	WY11609_00 AT  %MX11636.0 : BOOL; (*STN 5 PROCESS TANK VACUUM RELEASE AV5-2 (-161Y10) *)
	WY11609_01 AT  %MX11636.1 : BOOL; (*STN 5 PROCESS TANK VACUUM RELEASE AV5-2 (-161Y10) *)
	WY11609_02 AT  %MX11636.2 : BOOL; (*STN 5 PROCESS TANK VACUUM RELEASE AV5-2 (-161Y10) *)
	WY11609_03 AT  %MX11636.3 : BOOL; (*STN 5 PROCESS TANK VACUUM RELEASE AV5-2 (-161Y10) *)
	WY11609_04 AT  %MX11636.4 : BOOL; (*STN 5 PROCESS TANK VACUUM RELEASE AV5-2 (-161Y10) *)
	WY11609_05 AT  %MX11636.5 : BOOL; (*STN 5 PROCESS TANK VACUUM RELEASE AV5-2 (-161Y10) *)
	WY11609_06 AT  %MX11636.6 : BOOL; (*STN 5 PROCESS TANK VACUUM RELEASE AV5-2 (-161Y10) *)
	WY11609_07 AT  %MX11636.7 : BOOL; (*STN 5 PROCESS TANK VACUUM RELEASE AV5-2 (-161Y10) *)
	WY11609_08 AT  %MX11636.8 : BOOL; (*STN 5 PROCESS TANK VACUUM RELEASE AV5-2 (-161Y10) *)
	WY11609_09 AT  %MX11636.9 : BOOL; (*STN 5 PROCESS TANK VACUUM RELEASE AV5-2 (-161Y10) *)
	WY11609_10 AT  %MX11636.10 : BOOL; (*STN 5 PROCESS TANK VACUUM RELEASE AV5-2 (-161Y10) *)
	WY11609_11 AT  %MX11636.11 : BOOL; (*STN 5 PROCESS TANK VACUUM RELEASE AV5-2 (-161Y10) *)
	WY11609_12 AT  %MX11636.12 : BOOL; (*STN 5 PROCESS TANK VACUUM RELEASE AV5-2 (-161Y10) *)
	WY11609_13 AT  %MX11636.13 : BOOL; (*STN 5 PROCESS TANK VACUUM RELEASE AV5-2 (-161Y10) *)
	WY11609_14 AT  %MX11636.14 : BOOL; (*STN 5 PROCESS TANK VACUUM RELEASE AV5-2 (-161Y10) *)
	WY11609_15 AT  %MX11636.15 : BOOL; (*STN 5 PROCESS TANK VACUUM RELEASE AV5-2 (-161Y10) *)
	WY11609_16 AT  %MX11636.16 : BOOL; (*STN 5 PROCESS TANK VACUUM RELEASE AV5-2 (-161Y10) *)
	WY11609_17 AT  %MX11636.17 : BOOL; (*STN 5 PROCESS TANK VACUUM RELEASE AV5-2 (-161Y10) *)
	WY11609_18 AT  %MX11636.18 : BOOL; (*STN 5 PROCESS TANK VACUUM RELEASE AV5-2 (-161Y10) *)
	WY11609_19 AT  %MX11636.19 : BOOL; (*STN 5 PROCESS TANK VACUUM RELEASE AV5-2 (-161Y10) *)
	WY11609_20 AT  %MX11636.20 : BOOL; (*STN 5 PROCESS TANK VACUUM RELEASE AV5-2 (-161Y10) *)
	WY11609_21 AT  %MX11636.21 : BOOL; (*STN 5 PROCESS TANK VACUUM RELEASE AV5-2 (-161Y10) *)
	WY11609_22 AT  %MX11636.22 : BOOL; (*STN 5 PROCESS TANK VACUUM RELEASE AV5-2 (-161Y10) *)
	WY11609_23 AT  %MX11636.23 : BOOL; (*STN 5 PROCESS TANK VACUUM RELEASE AV5-2 (-161Y10) *)
	WY11609_24 AT  %MX11636.24 : BOOL; (*STN 5 PROCESS TANK VACUUM RELEASE AV5-2 (-161Y10) *)
	WY11609_25 AT  %MX11636.25 : BOOL; (*STN 5 PROCESS TANK VACUUM RELEASE AV5-2 (-161Y10) *)
	WY11609_26 AT  %MX11636.26 : BOOL; (*STN 5 PROCESS TANK VACUUM RELEASE AV5-2 (-161Y10) *)
	WY11609_27 AT  %MX11636.27 : BOOL; (*STN 5 PROCESS TANK VACUUM RELEASE AV5-2 (-161Y10) *)
	WY11609_28 AT  %MX11636.28 : BOOL; (*STN 5 PROCESS TANK VACUUM RELEASE AV5-2 (-161Y10) *)
	WY11609_29 AT  %MX11636.29 : BOOL; (*STN 5 PROCESS TANK VACUUM RELEASE AV5-2 (-161Y10) *)
	WY11609_30 AT  %MX11636.30 : BOOL; (*STN 5 PROCESS TANK VACUUM RELEASE AV5-2 (-161Y10) *)
	WY11609_31 AT  %MX11636.31 : BOOL; (*STN 5 PROCESS TANK VACUUM RELEASE AV5-2 (-161Y10) *)

	WY11610_00 AT  %MX11640.0 : BOOL; (*STN 5 BLOWER PROTECTION BUTTLEFLY AV5-3 (-161Y11) *)
	WY11610_01 AT  %MX11640.1 : BOOL; (*STN 5 BLOWER PROTECTION BUTTLEFLY AV5-3 (-161Y11) *)
	WY11610_02 AT  %MX11640.2 : BOOL; (*STN 5 BLOWER PROTECTION BUTTLEFLY AV5-3 (-161Y11) *)
	WY11610_03 AT  %MX11640.3 : BOOL; (*STN 5 BLOWER PROTECTION BUTTLEFLY AV5-3 (-161Y11) *)
	WY11610_04 AT  %MX11640.4 : BOOL; (*STN 5 BLOWER PROTECTION BUTTLEFLY AV5-3 (-161Y11) *)
	WY11610_05 AT  %MX11640.5 : BOOL; (*STN 5 BLOWER PROTECTION BUTTLEFLY AV5-3 (-161Y11) *)
	WY11610_06 AT  %MX11640.6 : BOOL; (*STN 5 BLOWER PROTECTION BUTTLEFLY AV5-3 (-161Y11) *)
	WY11610_07 AT  %MX11640.7 : BOOL; (*STN 5 BLOWER PROTECTION BUTTLEFLY AV5-3 (-161Y11) *)
	WY11610_08 AT  %MX11640.8 : BOOL; (*STN 5 BLOWER PROTECTION BUTTLEFLY AV5-3 (-161Y11) *)
	WY11610_09 AT  %MX11640.9 : BOOL; (*STN 5 BLOWER PROTECTION BUTTLEFLY AV5-3 (-161Y11) *)
	WY11610_10 AT  %MX11640.10 : BOOL; (*STN 5 BLOWER PROTECTION BUTTLEFLY AV5-3 (-161Y11) *)
	WY11610_11 AT  %MX11640.11 : BOOL; (*STN 5 BLOWER PROTECTION BUTTLEFLY AV5-3 (-161Y11) *)
	WY11610_12 AT  %MX11640.12 : BOOL; (*STN 5 BLOWER PROTECTION BUTTLEFLY AV5-3 (-161Y11) *)
	WY11610_13 AT  %MX11640.13 : BOOL; (*STN 5 BLOWER PROTECTION BUTTLEFLY AV5-3 (-161Y11) *)
	WY11610_14 AT  %MX11640.14 : BOOL; (*STN 5 BLOWER PROTECTION BUTTLEFLY AV5-3 (-161Y11) *)
	WY11610_15 AT  %MX11640.15 : BOOL; (*STN 5 BLOWER PROTECTION BUTTLEFLY AV5-3 (-161Y11) *)
	WY11610_16 AT  %MX11640.16 : BOOL; (*STN 5 BLOWER PROTECTION BUTTLEFLY AV5-3 (-161Y11) *)
	WY11610_17 AT  %MX11640.17 : BOOL; (*STN 5 BLOWER PROTECTION BUTTLEFLY AV5-3 (-161Y11) *)
	WY11610_18 AT  %MX11640.18 : BOOL; (*STN 5 BLOWER PROTECTION BUTTLEFLY AV5-3 (-161Y11) *)
	WY11610_19 AT  %MX11640.19 : BOOL; (*STN 5 BLOWER PROTECTION BUTTLEFLY AV5-3 (-161Y11) *)
	WY11610_20 AT  %MX11640.20 : BOOL; (*STN 5 BLOWER PROTECTION BUTTLEFLY AV5-3 (-161Y11) *)
	WY11610_21 AT  %MX11640.21 : BOOL; (*STN 5 BLOWER PROTECTION BUTTLEFLY AV5-3 (-161Y11) *)
	WY11610_22 AT  %MX11640.22 : BOOL; (*STN 5 BLOWER PROTECTION BUTTLEFLY AV5-3 (-161Y11) *)
	WY11610_23 AT  %MX11640.23 : BOOL; (*STN 5 BLOWER PROTECTION BUTTLEFLY AV5-3 (-161Y11) *)
	WY11610_24 AT  %MX11640.24 : BOOL; (*STN 5 BLOWER PROTECTION BUTTLEFLY AV5-3 (-161Y11) *)
	WY11610_25 AT  %MX11640.25 : BOOL; (*STN 5 BLOWER PROTECTION BUTTLEFLY AV5-3 (-161Y11) *)
	WY11610_26 AT  %MX11640.26 : BOOL; (*STN 5 BLOWER PROTECTION BUTTLEFLY AV5-3 (-161Y11) *)
	WY11610_27 AT  %MX11640.27 : BOOL; (*STN 5 BLOWER PROTECTION BUTTLEFLY AV5-3 (-161Y11) *)
	WY11610_28 AT  %MX11640.28 : BOOL; (*STN 5 BLOWER PROTECTION BUTTLEFLY AV5-3 (-161Y11) *)
	WY11610_29 AT  %MX11640.29 : BOOL; (*STN 5 BLOWER PROTECTION BUTTLEFLY AV5-3 (-161Y11) *)
	WY11610_30 AT  %MX11640.30 : BOOL; (*STN 5 BLOWER PROTECTION BUTTLEFLY AV5-3 (-161Y11) *)
	WY11610_31 AT  %MX11640.31 : BOOL; (*STN 5 BLOWER PROTECTION BUTTLEFLY AV5-3 (-161Y11) *)

	WY11611_00 AT  %MX11644.0 : BOOL; (*STN 5 BLOWER PROTECTION BUTTLEFLY AV5-4 (-161Y12) *)
	WY11611_01 AT  %MX11644.1 : BOOL; (*STN 5 BLOWER PROTECTION BUTTLEFLY AV5-4 (-161Y12) *)
	WY11611_02 AT  %MX11644.2 : BOOL; (*STN 5 BLOWER PROTECTION BUTTLEFLY AV5-4 (-161Y12) *)
	WY11611_03 AT  %MX11644.3 : BOOL; (*STN 5 BLOWER PROTECTION BUTTLEFLY AV5-4 (-161Y12) *)
	WY11611_04 AT  %MX11644.4 : BOOL; (*STN 5 BLOWER PROTECTION BUTTLEFLY AV5-4 (-161Y12) *)
	WY11611_05 AT  %MX11644.5 : BOOL; (*STN 5 BLOWER PROTECTION BUTTLEFLY AV5-4 (-161Y12) *)
	WY11611_06 AT  %MX11644.6 : BOOL; (*STN 5 BLOWER PROTECTION BUTTLEFLY AV5-4 (-161Y12) *)
	WY11611_07 AT  %MX11644.7 : BOOL; (*STN 5 BLOWER PROTECTION BUTTLEFLY AV5-4 (-161Y12) *)
	WY11611_08 AT  %MX11644.8 : BOOL; (*STN 5 BLOWER PROTECTION BUTTLEFLY AV5-4 (-161Y12) *)
	WY11611_09 AT  %MX11644.9 : BOOL; (*STN 5 BLOWER PROTECTION BUTTLEFLY AV5-4 (-161Y12) *)
	WY11611_10 AT  %MX11644.10 : BOOL; (*STN 5 BLOWER PROTECTION BUTTLEFLY AV5-4 (-161Y12) *)
	WY11611_11 AT  %MX11644.11 : BOOL; (*STN 5 BLOWER PROTECTION BUTTLEFLY AV5-4 (-161Y12) *)
	WY11611_12 AT  %MX11644.12 : BOOL; (*STN 5 BLOWER PROTECTION BUTTLEFLY AV5-4 (-161Y12) *)
	WY11611_13 AT  %MX11644.13 : BOOL; (*STN 5 BLOWER PROTECTION BUTTLEFLY AV5-4 (-161Y12) *)
	WY11611_14 AT  %MX11644.14 : BOOL; (*STN 5 BLOWER PROTECTION BUTTLEFLY AV5-4 (-161Y12) *)
	WY11611_15 AT  %MX11644.15 : BOOL; (*STN 5 BLOWER PROTECTION BUTTLEFLY AV5-4 (-161Y12) *)
	WY11611_16 AT  %MX11644.16 : BOOL; (*STN 5 BLOWER PROTECTION BUTTLEFLY AV5-4 (-161Y12) *)
	WY11611_17 AT  %MX11644.17 : BOOL; (*STN 5 BLOWER PROTECTION BUTTLEFLY AV5-4 (-161Y12) *)
	WY11611_18 AT  %MX11644.18 : BOOL; (*STN 5 BLOWER PROTECTION BUTTLEFLY AV5-4 (-161Y12) *)
	WY11611_19 AT  %MX11644.19 : BOOL; (*STN 5 BLOWER PROTECTION BUTTLEFLY AV5-4 (-161Y12) *)
	WY11611_20 AT  %MX11644.20 : BOOL; (*STN 5 BLOWER PROTECTION BUTTLEFLY AV5-4 (-161Y12) *)
	WY11611_21 AT  %MX11644.21 : BOOL; (*STN 5 BLOWER PROTECTION BUTTLEFLY AV5-4 (-161Y12) *)
	WY11611_22 AT  %MX11644.22 : BOOL; (*STN 5 BLOWER PROTECTION BUTTLEFLY AV5-4 (-161Y12) *)
	WY11611_23 AT  %MX11644.23 : BOOL; (*STN 5 BLOWER PROTECTION BUTTLEFLY AV5-4 (-161Y12) *)
	WY11611_24 AT  %MX11644.24 : BOOL; (*STN 5 BLOWER PROTECTION BUTTLEFLY AV5-4 (-161Y12) *)
	WY11611_25 AT  %MX11644.25 : BOOL; (*STN 5 BLOWER PROTECTION BUTTLEFLY AV5-4 (-161Y12) *)
	WY11611_26 AT  %MX11644.26 : BOOL; (*STN 5 BLOWER PROTECTION BUTTLEFLY AV5-4 (-161Y12) *)
	WY11611_27 AT  %MX11644.27 : BOOL; (*STN 5 BLOWER PROTECTION BUTTLEFLY AV5-4 (-161Y12) *)
	WY11611_28 AT  %MX11644.28 : BOOL; (*STN 5 BLOWER PROTECTION BUTTLEFLY AV5-4 (-161Y12) *)
	WY11611_29 AT  %MX11644.29 : BOOL; (*STN 5 BLOWER PROTECTION BUTTLEFLY AV5-4 (-161Y12) *)
	WY11611_30 AT  %MX11644.30 : BOOL; (*STN 5 BLOWER PROTECTION BUTTLEFLY AV5-4 (-161Y12) *)
	WY11611_31 AT  %MX11644.31 : BOOL; (*STN 5 BLOWER PROTECTION BUTTLEFLY AV5-4 (-161Y12) *)

	WY11612_00 AT  %MX11648.0 : BOOL; (*FACILITY CHILL WATER SUPPLY AV5-5 (-161Y13) *)
	WY11612_01 AT  %MX11648.1 : BOOL; (*FACILITY CHILL WATER SUPPLY AV5-5 (-161Y13) *)
	WY11612_02 AT  %MX11648.2 : BOOL; (*FACILITY CHILL WATER SUPPLY AV5-5 (-161Y13) *)
	WY11612_03 AT  %MX11648.3 : BOOL; (*FACILITY CHILL WATER SUPPLY AV5-5 (-161Y13) *)
	WY11612_04 AT  %MX11648.4 : BOOL; (*FACILITY CHILL WATER SUPPLY AV5-5 (-161Y13) *)
	WY11612_05 AT  %MX11648.5 : BOOL; (*FACILITY CHILL WATER SUPPLY AV5-5 (-161Y13) *)
	WY11612_06 AT  %MX11648.6 : BOOL; (*FACILITY CHILL WATER SUPPLY AV5-5 (-161Y13) *)
	WY11612_07 AT  %MX11648.7 : BOOL; (*FACILITY CHILL WATER SUPPLY AV5-5 (-161Y13) *)
	WY11612_08 AT  %MX11648.8 : BOOL; (*FACILITY CHILL WATER SUPPLY AV5-5 (-161Y13) *)
	WY11612_09 AT  %MX11648.9 : BOOL; (*FACILITY CHILL WATER SUPPLY AV5-5 (-161Y13) *)
	WY11612_10 AT  %MX11648.10 : BOOL; (*FACILITY CHILL WATER SUPPLY AV5-5 (-161Y13) *)
	WY11612_11 AT  %MX11648.11 : BOOL; (*FACILITY CHILL WATER SUPPLY AV5-5 (-161Y13) *)
	WY11612_12 AT  %MX11648.12 : BOOL; (*FACILITY CHILL WATER SUPPLY AV5-5 (-161Y13) *)
	WY11612_13 AT  %MX11648.13 : BOOL; (*FACILITY CHILL WATER SUPPLY AV5-5 (-161Y13) *)
	WY11612_14 AT  %MX11648.14 : BOOL; (*FACILITY CHILL WATER SUPPLY AV5-5 (-161Y13) *)
	WY11612_15 AT  %MX11648.15 : BOOL; (*FACILITY CHILL WATER SUPPLY AV5-5 (-161Y13) *)
	WY11612_16 AT  %MX11648.16 : BOOL; (*FACILITY CHILL WATER SUPPLY AV5-5 (-161Y13) *)
	WY11612_17 AT  %MX11648.17 : BOOL; (*FACILITY CHILL WATER SUPPLY AV5-5 (-161Y13) *)
	WY11612_18 AT  %MX11648.18 : BOOL; (*FACILITY CHILL WATER SUPPLY AV5-5 (-161Y13) *)
	WY11612_19 AT  %MX11648.19 : BOOL; (*FACILITY CHILL WATER SUPPLY AV5-5 (-161Y13) *)
	WY11612_20 AT  %MX11648.20 : BOOL; (*FACILITY CHILL WATER SUPPLY AV5-5 (-161Y13) *)
	WY11612_21 AT  %MX11648.21 : BOOL; (*FACILITY CHILL WATER SUPPLY AV5-5 (-161Y13) *)
	WY11612_22 AT  %MX11648.22 : BOOL; (*FACILITY CHILL WATER SUPPLY AV5-5 (-161Y13) *)
	WY11612_23 AT  %MX11648.23 : BOOL; (*FACILITY CHILL WATER SUPPLY AV5-5 (-161Y13) *)
	WY11612_24 AT  %MX11648.24 : BOOL; (*FACILITY CHILL WATER SUPPLY AV5-5 (-161Y13) *)
	WY11612_25 AT  %MX11648.25 : BOOL; (*FACILITY CHILL WATER SUPPLY AV5-5 (-161Y13) *)
	WY11612_26 AT  %MX11648.26 : BOOL; (*FACILITY CHILL WATER SUPPLY AV5-5 (-161Y13) *)
	WY11612_27 AT  %MX11648.27 : BOOL; (*FACILITY CHILL WATER SUPPLY AV5-5 (-161Y13) *)
	WY11612_28 AT  %MX11648.28 : BOOL; (*FACILITY CHILL WATER SUPPLY AV5-5 (-161Y13) *)
	WY11612_29 AT  %MX11648.29 : BOOL; (*FACILITY CHILL WATER SUPPLY AV5-5 (-161Y13) *)
	WY11612_30 AT  %MX11648.30 : BOOL; (*FACILITY CHILL WATER SUPPLY AV5-5 (-161Y13) *)
	WY11612_31 AT  %MX11648.31 : BOOL; (*FACILITY CHILL WATER SUPPLY AV5-5 (-161Y13) *)

	WY11613_00 AT  %MX11652.0 : BOOL; (*STN 4 & UNLOADING IONIZER CDA DISCHARGE AVION-1 (-161Y14,15) *)
	WY11613_01 AT  %MX11652.1 : BOOL; (*STN 4 & UNLOADING IONIZER CDA DISCHARGE AVION-1 (-161Y14,15) *)
	WY11613_02 AT  %MX11652.2 : BOOL; (*STN 4 & UNLOADING IONIZER CDA DISCHARGE AVION-1 (-161Y14,15) *)
	WY11613_03 AT  %MX11652.3 : BOOL; (*STN 4 & UNLOADING IONIZER CDA DISCHARGE AVION-1 (-161Y14,15) *)
	WY11613_04 AT  %MX11652.4 : BOOL; (*STN 4 & UNLOADING IONIZER CDA DISCHARGE AVION-1 (-161Y14,15) *)
	WY11613_05 AT  %MX11652.5 : BOOL; (*STN 4 & UNLOADING IONIZER CDA DISCHARGE AVION-1 (-161Y14,15) *)
	WY11613_06 AT  %MX11652.6 : BOOL; (*STN 4 & UNLOADING IONIZER CDA DISCHARGE AVION-1 (-161Y14,15) *)
	WY11613_07 AT  %MX11652.7 : BOOL; (*STN 4 & UNLOADING IONIZER CDA DISCHARGE AVION-1 (-161Y14,15) *)
	WY11613_08 AT  %MX11652.8 : BOOL; (*STN 4 & UNLOADING IONIZER CDA DISCHARGE AVION-1 (-161Y14,15) *)
	WY11613_09 AT  %MX11652.9 : BOOL; (*STN 4 & UNLOADING IONIZER CDA DISCHARGE AVION-1 (-161Y14,15) *)
	WY11613_10 AT  %MX11652.10 : BOOL; (*STN 4 & UNLOADING IONIZER CDA DISCHARGE AVION-1 (-161Y14,15) *)
	WY11613_11 AT  %MX11652.11 : BOOL; (*STN 4 & UNLOADING IONIZER CDA DISCHARGE AVION-1 (-161Y14,15) *)
	WY11613_12 AT  %MX11652.12 : BOOL; (*STN 4 & UNLOADING IONIZER CDA DISCHARGE AVION-1 (-161Y14,15) *)
	WY11613_13 AT  %MX11652.13 : BOOL; (*STN 4 & UNLOADING IONIZER CDA DISCHARGE AVION-1 (-161Y14,15) *)
	WY11613_14 AT  %MX11652.14 : BOOL; (*STN 4 & UNLOADING IONIZER CDA DISCHARGE AVION-1 (-161Y14,15) *)
	WY11613_15 AT  %MX11652.15 : BOOL; (*STN 4 & UNLOADING IONIZER CDA DISCHARGE AVION-1 (-161Y14,15) *)
	WY11613_16 AT  %MX11652.16 : BOOL; (*STN 4 & UNLOADING IONIZER CDA DISCHARGE AVION-1 (-161Y14,15) *)
	WY11613_17 AT  %MX11652.17 : BOOL; (*STN 4 & UNLOADING IONIZER CDA DISCHARGE AVION-1 (-161Y14,15) *)
	WY11613_18 AT  %MX11652.18 : BOOL; (*STN 4 & UNLOADING IONIZER CDA DISCHARGE AVION-1 (-161Y14,15) *)
	WY11613_19 AT  %MX11652.19 : BOOL; (*STN 4 & UNLOADING IONIZER CDA DISCHARGE AVION-1 (-161Y14,15) *)
	WY11613_20 AT  %MX11652.20 : BOOL; (*STN 4 & UNLOADING IONIZER CDA DISCHARGE AVION-1 (-161Y14,15) *)
	WY11613_21 AT  %MX11652.21 : BOOL; (*STN 4 & UNLOADING IONIZER CDA DISCHARGE AVION-1 (-161Y14,15) *)
	WY11613_22 AT  %MX11652.22 : BOOL; (*STN 4 & UNLOADING IONIZER CDA DISCHARGE AVION-1 (-161Y14,15) *)
	WY11613_23 AT  %MX11652.23 : BOOL; (*STN 4 & UNLOADING IONIZER CDA DISCHARGE AVION-1 (-161Y14,15) *)
	WY11613_24 AT  %MX11652.24 : BOOL; (*STN 4 & UNLOADING IONIZER CDA DISCHARGE AVION-1 (-161Y14,15) *)
	WY11613_25 AT  %MX11652.25 : BOOL; (*STN 4 & UNLOADING IONIZER CDA DISCHARGE AVION-1 (-161Y14,15) *)
	WY11613_26 AT  %MX11652.26 : BOOL; (*STN 4 & UNLOADING IONIZER CDA DISCHARGE AVION-1 (-161Y14,15) *)
	WY11613_27 AT  %MX11652.27 : BOOL; (*STN 4 & UNLOADING IONIZER CDA DISCHARGE AVION-1 (-161Y14,15) *)
	WY11613_28 AT  %MX11652.28 : BOOL; (*STN 4 & UNLOADING IONIZER CDA DISCHARGE AVION-1 (-161Y14,15) *)
	WY11613_29 AT  %MX11652.29 : BOOL; (*STN 4 & UNLOADING IONIZER CDA DISCHARGE AVION-1 (-161Y14,15) *)
	WY11613_30 AT  %MX11652.30 : BOOL; (*STN 4 & UNLOADING IONIZER CDA DISCHARGE AVION-1 (-161Y14,15) *)
	WY11613_31 AT  %MX11652.31 : BOOL; (*STN 4 & UNLOADING IONIZER CDA DISCHARGE AVION-1 (-161Y14,15) *)

	WY11614_00 AT  %MX11656.0 : BOOL; (*STN 4 IONIZER STATIC ELIMINATION STOP SIGNAL (-161U1) *)
	WY11614_01 AT  %MX11656.1 : BOOL; (*STN 4 IONIZER STATIC ELIMINATION STOP SIGNAL (-161U1) *)
	WY11614_02 AT  %MX11656.2 : BOOL; (*STN 4 IONIZER STATIC ELIMINATION STOP SIGNAL (-161U1) *)
	WY11614_03 AT  %MX11656.3 : BOOL; (*STN 4 IONIZER STATIC ELIMINATION STOP SIGNAL (-161U1) *)
	WY11614_04 AT  %MX11656.4 : BOOL; (*STN 4 IONIZER STATIC ELIMINATION STOP SIGNAL (-161U1) *)
	WY11614_05 AT  %MX11656.5 : BOOL; (*STN 4 IONIZER STATIC ELIMINATION STOP SIGNAL (-161U1) *)
	WY11614_06 AT  %MX11656.6 : BOOL; (*STN 4 IONIZER STATIC ELIMINATION STOP SIGNAL (-161U1) *)
	WY11614_07 AT  %MX11656.7 : BOOL; (*STN 4 IONIZER STATIC ELIMINATION STOP SIGNAL (-161U1) *)
	WY11614_08 AT  %MX11656.8 : BOOL; (*STN 4 IONIZER STATIC ELIMINATION STOP SIGNAL (-161U1) *)
	WY11614_09 AT  %MX11656.9 : BOOL; (*STN 4 IONIZER STATIC ELIMINATION STOP SIGNAL (-161U1) *)
	WY11614_10 AT  %MX11656.10 : BOOL; (*STN 4 IONIZER STATIC ELIMINATION STOP SIGNAL (-161U1) *)
	WY11614_11 AT  %MX11656.11 : BOOL; (*STN 4 IONIZER STATIC ELIMINATION STOP SIGNAL (-161U1) *)
	WY11614_12 AT  %MX11656.12 : BOOL; (*STN 4 IONIZER STATIC ELIMINATION STOP SIGNAL (-161U1) *)
	WY11614_13 AT  %MX11656.13 : BOOL; (*STN 4 IONIZER STATIC ELIMINATION STOP SIGNAL (-161U1) *)
	WY11614_14 AT  %MX11656.14 : BOOL; (*STN 4 IONIZER STATIC ELIMINATION STOP SIGNAL (-161U1) *)
	WY11614_15 AT  %MX11656.15 : BOOL; (*STN 4 IONIZER STATIC ELIMINATION STOP SIGNAL (-161U1) *)
	WY11614_16 AT  %MX11656.16 : BOOL; (*STN 4 IONIZER STATIC ELIMINATION STOP SIGNAL (-161U1) *)
	WY11614_17 AT  %MX11656.17 : BOOL; (*STN 4 IONIZER STATIC ELIMINATION STOP SIGNAL (-161U1) *)
	WY11614_18 AT  %MX11656.18 : BOOL; (*STN 4 IONIZER STATIC ELIMINATION STOP SIGNAL (-161U1) *)
	WY11614_19 AT  %MX11656.19 : BOOL; (*STN 4 IONIZER STATIC ELIMINATION STOP SIGNAL (-161U1) *)
	WY11614_20 AT  %MX11656.20 : BOOL; (*STN 4 IONIZER STATIC ELIMINATION STOP SIGNAL (-161U1) *)
	WY11614_21 AT  %MX11656.21 : BOOL; (*STN 4 IONIZER STATIC ELIMINATION STOP SIGNAL (-161U1) *)
	WY11614_22 AT  %MX11656.22 : BOOL; (*STN 4 IONIZER STATIC ELIMINATION STOP SIGNAL (-161U1) *)
	WY11614_23 AT  %MX11656.23 : BOOL; (*STN 4 IONIZER STATIC ELIMINATION STOP SIGNAL (-161U1) *)
	WY11614_24 AT  %MX11656.24 : BOOL; (*STN 4 IONIZER STATIC ELIMINATION STOP SIGNAL (-161U1) *)
	WY11614_25 AT  %MX11656.25 : BOOL; (*STN 4 IONIZER STATIC ELIMINATION STOP SIGNAL (-161U1) *)
	WY11614_26 AT  %MX11656.26 : BOOL; (*STN 4 IONIZER STATIC ELIMINATION STOP SIGNAL (-161U1) *)
	WY11614_27 AT  %MX11656.27 : BOOL; (*STN 4 IONIZER STATIC ELIMINATION STOP SIGNAL (-161U1) *)
	WY11614_28 AT  %MX11656.28 : BOOL; (*STN 4 IONIZER STATIC ELIMINATION STOP SIGNAL (-161U1) *)
	WY11614_29 AT  %MX11656.29 : BOOL; (*STN 4 IONIZER STATIC ELIMINATION STOP SIGNAL (-161U1) *)
	WY11614_30 AT  %MX11656.30 : BOOL; (*STN 4 IONIZER STATIC ELIMINATION STOP SIGNAL (-161U1) *)
	WY11614_31 AT  %MX11656.31 : BOOL; (*STN 4 IONIZER STATIC ELIMINATION STOP SIGNAL (-161U1) *)

	WY11615_00 AT  %MX11660.0 : BOOL; (*UNLOADING IONIZER STATIC ELIMINATION STOP SIGNAL (-161U2) *)
	WY11615_01 AT  %MX11660.1 : BOOL; (*UNLOADING IONIZER STATIC ELIMINATION STOP SIGNAL (-161U2) *)
	WY11615_02 AT  %MX11660.2 : BOOL; (*UNLOADING IONIZER STATIC ELIMINATION STOP SIGNAL (-161U2) *)
	WY11615_03 AT  %MX11660.3 : BOOL; (*UNLOADING IONIZER STATIC ELIMINATION STOP SIGNAL (-161U2) *)
	WY11615_04 AT  %MX11660.4 : BOOL; (*UNLOADING IONIZER STATIC ELIMINATION STOP SIGNAL (-161U2) *)
	WY11615_05 AT  %MX11660.5 : BOOL; (*UNLOADING IONIZER STATIC ELIMINATION STOP SIGNAL (-161U2) *)
	WY11615_06 AT  %MX11660.6 : BOOL; (*UNLOADING IONIZER STATIC ELIMINATION STOP SIGNAL (-161U2) *)
	WY11615_07 AT  %MX11660.7 : BOOL; (*UNLOADING IONIZER STATIC ELIMINATION STOP SIGNAL (-161U2) *)
	WY11615_08 AT  %MX11660.8 : BOOL; (*UNLOADING IONIZER STATIC ELIMINATION STOP SIGNAL (-161U2) *)
	WY11615_09 AT  %MX11660.9 : BOOL; (*UNLOADING IONIZER STATIC ELIMINATION STOP SIGNAL (-161U2) *)
	WY11615_10 AT  %MX11660.10 : BOOL; (*UNLOADING IONIZER STATIC ELIMINATION STOP SIGNAL (-161U2) *)
	WY11615_11 AT  %MX11660.11 : BOOL; (*UNLOADING IONIZER STATIC ELIMINATION STOP SIGNAL (-161U2) *)
	WY11615_12 AT  %MX11660.12 : BOOL; (*UNLOADING IONIZER STATIC ELIMINATION STOP SIGNAL (-161U2) *)
	WY11615_13 AT  %MX11660.13 : BOOL; (*UNLOADING IONIZER STATIC ELIMINATION STOP SIGNAL (-161U2) *)
	WY11615_14 AT  %MX11660.14 : BOOL; (*UNLOADING IONIZER STATIC ELIMINATION STOP SIGNAL (-161U2) *)
	WY11615_15 AT  %MX11660.15 : BOOL; (*UNLOADING IONIZER STATIC ELIMINATION STOP SIGNAL (-161U2) *)
	WY11615_16 AT  %MX11660.16 : BOOL; (*UNLOADING IONIZER STATIC ELIMINATION STOP SIGNAL (-161U2) *)
	WY11615_17 AT  %MX11660.17 : BOOL; (*UNLOADING IONIZER STATIC ELIMINATION STOP SIGNAL (-161U2) *)
	WY11615_18 AT  %MX11660.18 : BOOL; (*UNLOADING IONIZER STATIC ELIMINATION STOP SIGNAL (-161U2) *)
	WY11615_19 AT  %MX11660.19 : BOOL; (*UNLOADING IONIZER STATIC ELIMINATION STOP SIGNAL (-161U2) *)
	WY11615_20 AT  %MX11660.20 : BOOL; (*UNLOADING IONIZER STATIC ELIMINATION STOP SIGNAL (-161U2) *)
	WY11615_21 AT  %MX11660.21 : BOOL; (*UNLOADING IONIZER STATIC ELIMINATION STOP SIGNAL (-161U2) *)
	WY11615_22 AT  %MX11660.22 : BOOL; (*UNLOADING IONIZER STATIC ELIMINATION STOP SIGNAL (-161U2) *)
	WY11615_23 AT  %MX11660.23 : BOOL; (*UNLOADING IONIZER STATIC ELIMINATION STOP SIGNAL (-161U2) *)
	WY11615_24 AT  %MX11660.24 : BOOL; (*UNLOADING IONIZER STATIC ELIMINATION STOP SIGNAL (-161U2) *)
	WY11615_25 AT  %MX11660.25 : BOOL; (*UNLOADING IONIZER STATIC ELIMINATION STOP SIGNAL (-161U2) *)
	WY11615_26 AT  %MX11660.26 : BOOL; (*UNLOADING IONIZER STATIC ELIMINATION STOP SIGNAL (-161U2) *)
	WY11615_27 AT  %MX11660.27 : BOOL; (*UNLOADING IONIZER STATIC ELIMINATION STOP SIGNAL (-161U2) *)
	WY11615_28 AT  %MX11660.28 : BOOL; (*UNLOADING IONIZER STATIC ELIMINATION STOP SIGNAL (-161U2) *)
	WY11615_29 AT  %MX11660.29 : BOOL; (*UNLOADING IONIZER STATIC ELIMINATION STOP SIGNAL (-161U2) *)
	WY11615_30 AT  %MX11660.30 : BOOL; (*UNLOADING IONIZER STATIC ELIMINATION STOP SIGNAL (-161U2) *)
	WY11615_31 AT  %MX11660.31 : BOOL; (*UNLOADING IONIZER STATIC ELIMINATION STOP SIGNAL (-161U2) *)

	WY11700_00 AT  %MX11700.0 : BOOL; (*STN 4 CDA CYLINDER - IN (-162Y1) *)
	WY11700_01 AT  %MX11700.1 : BOOL; (*STN 4 CDA CYLINDER - IN (-162Y1) *)
	WY11700_02 AT  %MX11700.2 : BOOL; (*STN 4 CDA CYLINDER - IN (-162Y1) *)
	WY11700_03 AT  %MX11700.3 : BOOL; (*STN 4 CDA CYLINDER - IN (-162Y1) *)
	WY11700_04 AT  %MX11700.4 : BOOL; (*STN 4 CDA CYLINDER - IN (-162Y1) *)
	WY11700_05 AT  %MX11700.5 : BOOL; (*STN 4 CDA CYLINDER - IN (-162Y1) *)
	WY11700_06 AT  %MX11700.6 : BOOL; (*STN 4 CDA CYLINDER - IN (-162Y1) *)
	WY11700_07 AT  %MX11700.7 : BOOL; (*STN 4 CDA CYLINDER - IN (-162Y1) *)
	WY11700_08 AT  %MX11700.8 : BOOL; (*STN 4 CDA CYLINDER - IN (-162Y1) *)
	WY11700_09 AT  %MX11700.9 : BOOL; (*STN 4 CDA CYLINDER - IN (-162Y1) *)
	WY11700_10 AT  %MX11700.10 : BOOL; (*STN 4 CDA CYLINDER - IN (-162Y1) *)
	WY11700_11 AT  %MX11700.11 : BOOL; (*STN 4 CDA CYLINDER - IN (-162Y1) *)
	WY11700_12 AT  %MX11700.12 : BOOL; (*STN 4 CDA CYLINDER - IN (-162Y1) *)
	WY11700_13 AT  %MX11700.13 : BOOL; (*STN 4 CDA CYLINDER - IN (-162Y1) *)
	WY11700_14 AT  %MX11700.14 : BOOL; (*STN 4 CDA CYLINDER - IN (-162Y1) *)
	WY11700_15 AT  %MX11700.15 : BOOL; (*STN 4 CDA CYLINDER - IN (-162Y1) *)
	WY11700_16 AT  %MX11700.16 : BOOL; (*STN 4 CDA CYLINDER - IN (-162Y1) *)
	WY11700_17 AT  %MX11700.17 : BOOL; (*STN 4 CDA CYLINDER - IN (-162Y1) *)
	WY11700_18 AT  %MX11700.18 : BOOL; (*STN 4 CDA CYLINDER - IN (-162Y1) *)
	WY11700_19 AT  %MX11700.19 : BOOL; (*STN 4 CDA CYLINDER - IN (-162Y1) *)
	WY11700_20 AT  %MX11700.20 : BOOL; (*STN 4 CDA CYLINDER - IN (-162Y1) *)
	WY11700_21 AT  %MX11700.21 : BOOL; (*STN 4 CDA CYLINDER - IN (-162Y1) *)
	WY11700_22 AT  %MX11700.22 : BOOL; (*STN 4 CDA CYLINDER - IN (-162Y1) *)
	WY11700_23 AT  %MX11700.23 : BOOL; (*STN 4 CDA CYLINDER - IN (-162Y1) *)
	WY11700_24 AT  %MX11700.24 : BOOL; (*STN 4 CDA CYLINDER - IN (-162Y1) *)
	WY11700_25 AT  %MX11700.25 : BOOL; (*STN 4 CDA CYLINDER - IN (-162Y1) *)
	WY11700_26 AT  %MX11700.26 : BOOL; (*STN 4 CDA CYLINDER - IN (-162Y1) *)
	WY11700_27 AT  %MX11700.27 : BOOL; (*STN 4 CDA CYLINDER - IN (-162Y1) *)
	WY11700_28 AT  %MX11700.28 : BOOL; (*STN 4 CDA CYLINDER - IN (-162Y1) *)
	WY11700_29 AT  %MX11700.29 : BOOL; (*STN 4 CDA CYLINDER - IN (-162Y1) *)
	WY11700_30 AT  %MX11700.30 : BOOL; (*STN 4 CDA CYLINDER - IN (-162Y1) *)
	WY11700_31 AT  %MX11700.31 : BOOL; (*STN 4 CDA CYLINDER - IN (-162Y1) *)

	WY11701_00 AT  %MX11704.0 : BOOL; (*STN 4 CDA CYLINDER - OUT (-162Y2) *)
	WY11701_01 AT  %MX11704.1 : BOOL; (*STN 4 CDA CYLINDER - OUT (-162Y2) *)
	WY11701_02 AT  %MX11704.2 : BOOL; (*STN 4 CDA CYLINDER - OUT (-162Y2) *)
	WY11701_03 AT  %MX11704.3 : BOOL; (*STN 4 CDA CYLINDER - OUT (-162Y2) *)
	WY11701_04 AT  %MX11704.4 : BOOL; (*STN 4 CDA CYLINDER - OUT (-162Y2) *)
	WY11701_05 AT  %MX11704.5 : BOOL; (*STN 4 CDA CYLINDER - OUT (-162Y2) *)
	WY11701_06 AT  %MX11704.6 : BOOL; (*STN 4 CDA CYLINDER - OUT (-162Y2) *)
	WY11701_07 AT  %MX11704.7 : BOOL; (*STN 4 CDA CYLINDER - OUT (-162Y2) *)
	WY11701_08 AT  %MX11704.8 : BOOL; (*STN 4 CDA CYLINDER - OUT (-162Y2) *)
	WY11701_09 AT  %MX11704.9 : BOOL; (*STN 4 CDA CYLINDER - OUT (-162Y2) *)
	WY11701_10 AT  %MX11704.10 : BOOL; (*STN 4 CDA CYLINDER - OUT (-162Y2) *)
	WY11701_11 AT  %MX11704.11 : BOOL; (*STN 4 CDA CYLINDER - OUT (-162Y2) *)
	WY11701_12 AT  %MX11704.12 : BOOL; (*STN 4 CDA CYLINDER - OUT (-162Y2) *)
	WY11701_13 AT  %MX11704.13 : BOOL; (*STN 4 CDA CYLINDER - OUT (-162Y2) *)
	WY11701_14 AT  %MX11704.14 : BOOL; (*STN 4 CDA CYLINDER - OUT (-162Y2) *)
	WY11701_15 AT  %MX11704.15 : BOOL; (*STN 4 CDA CYLINDER - OUT (-162Y2) *)
	WY11701_16 AT  %MX11704.16 : BOOL; (*STN 4 CDA CYLINDER - OUT (-162Y2) *)
	WY11701_17 AT  %MX11704.17 : BOOL; (*STN 4 CDA CYLINDER - OUT (-162Y2) *)
	WY11701_18 AT  %MX11704.18 : BOOL; (*STN 4 CDA CYLINDER - OUT (-162Y2) *)
	WY11701_19 AT  %MX11704.19 : BOOL; (*STN 4 CDA CYLINDER - OUT (-162Y2) *)
	WY11701_20 AT  %MX11704.20 : BOOL; (*STN 4 CDA CYLINDER - OUT (-162Y2) *)
	WY11701_21 AT  %MX11704.21 : BOOL; (*STN 4 CDA CYLINDER - OUT (-162Y2) *)
	WY11701_22 AT  %MX11704.22 : BOOL; (*STN 4 CDA CYLINDER - OUT (-162Y2) *)
	WY11701_23 AT  %MX11704.23 : BOOL; (*STN 4 CDA CYLINDER - OUT (-162Y2) *)
	WY11701_24 AT  %MX11704.24 : BOOL; (*STN 4 CDA CYLINDER - OUT (-162Y2) *)
	WY11701_25 AT  %MX11704.25 : BOOL; (*STN 4 CDA CYLINDER - OUT (-162Y2) *)
	WY11701_26 AT  %MX11704.26 : BOOL; (*STN 4 CDA CYLINDER - OUT (-162Y2) *)
	WY11701_27 AT  %MX11704.27 : BOOL; (*STN 4 CDA CYLINDER - OUT (-162Y2) *)
	WY11701_28 AT  %MX11704.28 : BOOL; (*STN 4 CDA CYLINDER - OUT (-162Y2) *)
	WY11701_29 AT  %MX11704.29 : BOOL; (*STN 4 CDA CYLINDER - OUT (-162Y2) *)
	WY11701_30 AT  %MX11704.30 : BOOL; (*STN 4 CDA CYLINDER - OUT (-162Y2) *)
	WY11701_31 AT  %MX11704.31 : BOOL; (*STN 4 CDA CYLINDER - OUT (-162Y2) *)

	WY11702_00 AT  %MX11708.0 : BOOL; (*RAMP PUMP AV (-162Y3) *)
	WY11702_01 AT  %MX11708.1 : BOOL; (*RAMP PUMP AV (-162Y3) *)
	WY11702_02 AT  %MX11708.2 : BOOL; (*RAMP PUMP AV (-162Y3) *)
	WY11702_03 AT  %MX11708.3 : BOOL; (*RAMP PUMP AV (-162Y3) *)
	WY11702_04 AT  %MX11708.4 : BOOL; (*RAMP PUMP AV (-162Y3) *)
	WY11702_05 AT  %MX11708.5 : BOOL; (*RAMP PUMP AV (-162Y3) *)
	WY11702_06 AT  %MX11708.6 : BOOL; (*RAMP PUMP AV (-162Y3) *)
	WY11702_07 AT  %MX11708.7 : BOOL; (*RAMP PUMP AV (-162Y3) *)
	WY11702_08 AT  %MX11708.8 : BOOL; (*RAMP PUMP AV (-162Y3) *)
	WY11702_09 AT  %MX11708.9 : BOOL; (*RAMP PUMP AV (-162Y3) *)
	WY11702_10 AT  %MX11708.10 : BOOL; (*RAMP PUMP AV (-162Y3) *)
	WY11702_11 AT  %MX11708.11 : BOOL; (*RAMP PUMP AV (-162Y3) *)
	WY11702_12 AT  %MX11708.12 : BOOL; (*RAMP PUMP AV (-162Y3) *)
	WY11702_13 AT  %MX11708.13 : BOOL; (*RAMP PUMP AV (-162Y3) *)
	WY11702_14 AT  %MX11708.14 : BOOL; (*RAMP PUMP AV (-162Y3) *)
	WY11702_15 AT  %MX11708.15 : BOOL; (*RAMP PUMP AV (-162Y3) *)
	WY11702_16 AT  %MX11708.16 : BOOL; (*RAMP PUMP AV (-162Y3) *)
	WY11702_17 AT  %MX11708.17 : BOOL; (*RAMP PUMP AV (-162Y3) *)
	WY11702_18 AT  %MX11708.18 : BOOL; (*RAMP PUMP AV (-162Y3) *)
	WY11702_19 AT  %MX11708.19 : BOOL; (*RAMP PUMP AV (-162Y3) *)
	WY11702_20 AT  %MX11708.20 : BOOL; (*RAMP PUMP AV (-162Y3) *)
	WY11702_21 AT  %MX11708.21 : BOOL; (*RAMP PUMP AV (-162Y3) *)
	WY11702_22 AT  %MX11708.22 : BOOL; (*RAMP PUMP AV (-162Y3) *)
	WY11702_23 AT  %MX11708.23 : BOOL; (*RAMP PUMP AV (-162Y3) *)
	WY11702_24 AT  %MX11708.24 : BOOL; (*RAMP PUMP AV (-162Y3) *)
	WY11702_25 AT  %MX11708.25 : BOOL; (*RAMP PUMP AV (-162Y3) *)
	WY11702_26 AT  %MX11708.26 : BOOL; (*RAMP PUMP AV (-162Y3) *)
	WY11702_27 AT  %MX11708.27 : BOOL; (*RAMP PUMP AV (-162Y3) *)
	WY11702_28 AT  %MX11708.28 : BOOL; (*RAMP PUMP AV (-162Y3) *)
	WY11702_29 AT  %MX11708.29 : BOOL; (*RAMP PUMP AV (-162Y3) *)
	WY11702_30 AT  %MX11708.30 : BOOL; (*RAMP PUMP AV (-162Y3) *)
	WY11702_31 AT  %MX11708.31 : BOOL; (*RAMP PUMP AV (-162Y3) *)

	WY11703_00 AT  %MX11712.0 : BOOL; (*RESERVED *)
	WY11703_01 AT  %MX11712.1 : BOOL; (*RESERVED *)
	WY11703_02 AT  %MX11712.2 : BOOL; (*RESERVED *)
	WY11703_03 AT  %MX11712.3 : BOOL; (*RESERVED *)
	WY11703_04 AT  %MX11712.4 : BOOL; (*RESERVED *)
	WY11703_05 AT  %MX11712.5 : BOOL; (*RESERVED *)
	WY11703_06 AT  %MX11712.6 : BOOL; (*RESERVED *)
	WY11703_07 AT  %MX11712.7 : BOOL; (*RESERVED *)
	WY11703_08 AT  %MX11712.8 : BOOL; (*RESERVED *)
	WY11703_09 AT  %MX11712.9 : BOOL; (*RESERVED *)
	WY11703_10 AT  %MX11712.10 : BOOL; (*RESERVED *)
	WY11703_11 AT  %MX11712.11 : BOOL; (*RESERVED *)
	WY11703_12 AT  %MX11712.12 : BOOL; (*RESERVED *)
	WY11703_13 AT  %MX11712.13 : BOOL; (*RESERVED *)
	WY11703_14 AT  %MX11712.14 : BOOL; (*RESERVED *)
	WY11703_15 AT  %MX11712.15 : BOOL; (*RESERVED *)
	WY11703_16 AT  %MX11712.16 : BOOL; (*RESERVED *)
	WY11703_17 AT  %MX11712.17 : BOOL; (*RESERVED *)
	WY11703_18 AT  %MX11712.18 : BOOL; (*RESERVED *)
	WY11703_19 AT  %MX11712.19 : BOOL; (*RESERVED *)
	WY11703_20 AT  %MX11712.20 : BOOL; (*RESERVED *)
	WY11703_21 AT  %MX11712.21 : BOOL; (*RESERVED *)
	WY11703_22 AT  %MX11712.22 : BOOL; (*RESERVED *)
	WY11703_23 AT  %MX11712.23 : BOOL; (*RESERVED *)
	WY11703_24 AT  %MX11712.24 : BOOL; (*RESERVED *)
	WY11703_25 AT  %MX11712.25 : BOOL; (*RESERVED *)
	WY11703_26 AT  %MX11712.26 : BOOL; (*RESERVED *)
	WY11703_27 AT  %MX11712.27 : BOOL; (*RESERVED *)
	WY11703_28 AT  %MX11712.28 : BOOL; (*RESERVED *)
	WY11703_29 AT  %MX11712.29 : BOOL; (*RESERVED *)
	WY11703_30 AT  %MX11712.30 : BOOL; (*RESERVED *)
	WY11703_31 AT  %MX11712.31 : BOOL; (*RESERVED *)

	WY11704_00 AT  %MX11716.0 : BOOL; (*RESERVED *)
	WY11704_01 AT  %MX11716.1 : BOOL; (*RESERVED *)
	WY11704_02 AT  %MX11716.2 : BOOL; (*RESERVED *)
	WY11704_03 AT  %MX11716.3 : BOOL; (*RESERVED *)
	WY11704_04 AT  %MX11716.4 : BOOL; (*RESERVED *)
	WY11704_05 AT  %MX11716.5 : BOOL; (*RESERVED *)
	WY11704_06 AT  %MX11716.6 : BOOL; (*RESERVED *)
	WY11704_07 AT  %MX11716.7 : BOOL; (*RESERVED *)
	WY11704_08 AT  %MX11716.8 : BOOL; (*RESERVED *)
	WY11704_09 AT  %MX11716.9 : BOOL; (*RESERVED *)
	WY11704_10 AT  %MX11716.10 : BOOL; (*RESERVED *)
	WY11704_11 AT  %MX11716.11 : BOOL; (*RESERVED *)
	WY11704_12 AT  %MX11716.12 : BOOL; (*RESERVED *)
	WY11704_13 AT  %MX11716.13 : BOOL; (*RESERVED *)
	WY11704_14 AT  %MX11716.14 : BOOL; (*RESERVED *)
	WY11704_15 AT  %MX11716.15 : BOOL; (*RESERVED *)
	WY11704_16 AT  %MX11716.16 : BOOL; (*RESERVED *)
	WY11704_17 AT  %MX11716.17 : BOOL; (*RESERVED *)
	WY11704_18 AT  %MX11716.18 : BOOL; (*RESERVED *)
	WY11704_19 AT  %MX11716.19 : BOOL; (*RESERVED *)
	WY11704_20 AT  %MX11716.20 : BOOL; (*RESERVED *)
	WY11704_21 AT  %MX11716.21 : BOOL; (*RESERVED *)
	WY11704_22 AT  %MX11716.22 : BOOL; (*RESERVED *)
	WY11704_23 AT  %MX11716.23 : BOOL; (*RESERVED *)
	WY11704_24 AT  %MX11716.24 : BOOL; (*RESERVED *)
	WY11704_25 AT  %MX11716.25 : BOOL; (*RESERVED *)
	WY11704_26 AT  %MX11716.26 : BOOL; (*RESERVED *)
	WY11704_27 AT  %MX11716.27 : BOOL; (*RESERVED *)
	WY11704_28 AT  %MX11716.28 : BOOL; (*RESERVED *)
	WY11704_29 AT  %MX11716.29 : BOOL; (*RESERVED *)
	WY11704_30 AT  %MX11716.30 : BOOL; (*RESERVED *)
	WY11704_31 AT  %MX11716.31 : BOOL; (*RESERVED *)

	WY11705_00 AT  %MX11720.0 : BOOL; (*RESERVED *)
	WY11705_01 AT  %MX11720.1 : BOOL; (*RESERVED *)
	WY11705_02 AT  %MX11720.2 : BOOL; (*RESERVED *)
	WY11705_03 AT  %MX11720.3 : BOOL; (*RESERVED *)
	WY11705_04 AT  %MX11720.4 : BOOL; (*RESERVED *)
	WY11705_05 AT  %MX11720.5 : BOOL; (*RESERVED *)
	WY11705_06 AT  %MX11720.6 : BOOL; (*RESERVED *)
	WY11705_07 AT  %MX11720.7 : BOOL; (*RESERVED *)
	WY11705_08 AT  %MX11720.8 : BOOL; (*RESERVED *)
	WY11705_09 AT  %MX11720.9 : BOOL; (*RESERVED *)
	WY11705_10 AT  %MX11720.10 : BOOL; (*RESERVED *)
	WY11705_11 AT  %MX11720.11 : BOOL; (*RESERVED *)
	WY11705_12 AT  %MX11720.12 : BOOL; (*RESERVED *)
	WY11705_13 AT  %MX11720.13 : BOOL; (*RESERVED *)
	WY11705_14 AT  %MX11720.14 : BOOL; (*RESERVED *)
	WY11705_15 AT  %MX11720.15 : BOOL; (*RESERVED *)
	WY11705_16 AT  %MX11720.16 : BOOL; (*RESERVED *)
	WY11705_17 AT  %MX11720.17 : BOOL; (*RESERVED *)
	WY11705_18 AT  %MX11720.18 : BOOL; (*RESERVED *)
	WY11705_19 AT  %MX11720.19 : BOOL; (*RESERVED *)
	WY11705_20 AT  %MX11720.20 : BOOL; (*RESERVED *)
	WY11705_21 AT  %MX11720.21 : BOOL; (*RESERVED *)
	WY11705_22 AT  %MX11720.22 : BOOL; (*RESERVED *)
	WY11705_23 AT  %MX11720.23 : BOOL; (*RESERVED *)
	WY11705_24 AT  %MX11720.24 : BOOL; (*RESERVED *)
	WY11705_25 AT  %MX11720.25 : BOOL; (*RESERVED *)
	WY11705_26 AT  %MX11720.26 : BOOL; (*RESERVED *)
	WY11705_27 AT  %MX11720.27 : BOOL; (*RESERVED *)
	WY11705_28 AT  %MX11720.28 : BOOL; (*RESERVED *)
	WY11705_29 AT  %MX11720.29 : BOOL; (*RESERVED *)
	WY11705_30 AT  %MX11720.30 : BOOL; (*RESERVED *)
	WY11705_31 AT  %MX11720.31 : BOOL; (*RESERVED *)

	WY11706_00 AT  %MX11724.0 : BOOL; (*RESERVED *)
	WY11706_01 AT  %MX11724.1 : BOOL; (*RESERVED *)
	WY11706_02 AT  %MX11724.2 : BOOL; (*RESERVED *)
	WY11706_03 AT  %MX11724.3 : BOOL; (*RESERVED *)
	WY11706_04 AT  %MX11724.4 : BOOL; (*RESERVED *)
	WY11706_05 AT  %MX11724.5 : BOOL; (*RESERVED *)
	WY11706_06 AT  %MX11724.6 : BOOL; (*RESERVED *)
	WY11706_07 AT  %MX11724.7 : BOOL; (*RESERVED *)
	WY11706_08 AT  %MX11724.8 : BOOL; (*RESERVED *)
	WY11706_09 AT  %MX11724.9 : BOOL; (*RESERVED *)
	WY11706_10 AT  %MX11724.10 : BOOL; (*RESERVED *)
	WY11706_11 AT  %MX11724.11 : BOOL; (*RESERVED *)
	WY11706_12 AT  %MX11724.12 : BOOL; (*RESERVED *)
	WY11706_13 AT  %MX11724.13 : BOOL; (*RESERVED *)
	WY11706_14 AT  %MX11724.14 : BOOL; (*RESERVED *)
	WY11706_15 AT  %MX11724.15 : BOOL; (*RESERVED *)
	WY11706_16 AT  %MX11724.16 : BOOL; (*RESERVED *)
	WY11706_17 AT  %MX11724.17 : BOOL; (*RESERVED *)
	WY11706_18 AT  %MX11724.18 : BOOL; (*RESERVED *)
	WY11706_19 AT  %MX11724.19 : BOOL; (*RESERVED *)
	WY11706_20 AT  %MX11724.20 : BOOL; (*RESERVED *)
	WY11706_21 AT  %MX11724.21 : BOOL; (*RESERVED *)
	WY11706_22 AT  %MX11724.22 : BOOL; (*RESERVED *)
	WY11706_23 AT  %MX11724.23 : BOOL; (*RESERVED *)
	WY11706_24 AT  %MX11724.24 : BOOL; (*RESERVED *)
	WY11706_25 AT  %MX11724.25 : BOOL; (*RESERVED *)
	WY11706_26 AT  %MX11724.26 : BOOL; (*RESERVED *)
	WY11706_27 AT  %MX11724.27 : BOOL; (*RESERVED *)
	WY11706_28 AT  %MX11724.28 : BOOL; (*RESERVED *)
	WY11706_29 AT  %MX11724.29 : BOOL; (*RESERVED *)
	WY11706_30 AT  %MX11724.30 : BOOL; (*RESERVED *)
	WY11706_31 AT  %MX11724.31 : BOOL; (*RESERVED *)

	WY11707_00 AT  %MX11728.0 : BOOL; (*RESERVED *)
	WY11707_01 AT  %MX11728.1 : BOOL; (*RESERVED *)
	WY11707_02 AT  %MX11728.2 : BOOL; (*RESERVED *)
	WY11707_03 AT  %MX11728.3 : BOOL; (*RESERVED *)
	WY11707_04 AT  %MX11728.4 : BOOL; (*RESERVED *)
	WY11707_05 AT  %MX11728.5 : BOOL; (*RESERVED *)
	WY11707_06 AT  %MX11728.6 : BOOL; (*RESERVED *)
	WY11707_07 AT  %MX11728.7 : BOOL; (*RESERVED *)
	WY11707_08 AT  %MX11728.8 : BOOL; (*RESERVED *)
	WY11707_09 AT  %MX11728.9 : BOOL; (*RESERVED *)
	WY11707_10 AT  %MX11728.10 : BOOL; (*RESERVED *)
	WY11707_11 AT  %MX11728.11 : BOOL; (*RESERVED *)
	WY11707_12 AT  %MX11728.12 : BOOL; (*RESERVED *)
	WY11707_13 AT  %MX11728.13 : BOOL; (*RESERVED *)
	WY11707_14 AT  %MX11728.14 : BOOL; (*RESERVED *)
	WY11707_15 AT  %MX11728.15 : BOOL; (*RESERVED *)
	WY11707_16 AT  %MX11728.16 : BOOL; (*RESERVED *)
	WY11707_17 AT  %MX11728.17 : BOOL; (*RESERVED *)
	WY11707_18 AT  %MX11728.18 : BOOL; (*RESERVED *)
	WY11707_19 AT  %MX11728.19 : BOOL; (*RESERVED *)
	WY11707_20 AT  %MX11728.20 : BOOL; (*RESERVED *)
	WY11707_21 AT  %MX11728.21 : BOOL; (*RESERVED *)
	WY11707_22 AT  %MX11728.22 : BOOL; (*RESERVED *)
	WY11707_23 AT  %MX11728.23 : BOOL; (*RESERVED *)
	WY11707_24 AT  %MX11728.24 : BOOL; (*RESERVED *)
	WY11707_25 AT  %MX11728.25 : BOOL; (*RESERVED *)
	WY11707_26 AT  %MX11728.26 : BOOL; (*RESERVED *)
	WY11707_27 AT  %MX11728.27 : BOOL; (*RESERVED *)
	WY11707_28 AT  %MX11728.28 : BOOL; (*RESERVED *)
	WY11707_29 AT  %MX11728.29 : BOOL; (*RESERVED *)
	WY11707_30 AT  %MX11728.30 : BOOL; (*RESERVED *)
	WY11707_31 AT  %MX11728.31 : BOOL; (*RESERVED *)

	WY11708_00 AT  %MX11732.0 : BOOL; (*RESERVED *)
	WY11708_01 AT  %MX11732.1 : BOOL; (*RESERVED *)
	WY11708_02 AT  %MX11732.2 : BOOL; (*RESERVED *)
	WY11708_03 AT  %MX11732.3 : BOOL; (*RESERVED *)
	WY11708_04 AT  %MX11732.4 : BOOL; (*RESERVED *)
	WY11708_05 AT  %MX11732.5 : BOOL; (*RESERVED *)
	WY11708_06 AT  %MX11732.6 : BOOL; (*RESERVED *)
	WY11708_07 AT  %MX11732.7 : BOOL; (*RESERVED *)
	WY11708_08 AT  %MX11732.8 : BOOL; (*RESERVED *)
	WY11708_09 AT  %MX11732.9 : BOOL; (*RESERVED *)
	WY11708_10 AT  %MX11732.10 : BOOL; (*RESERVED *)
	WY11708_11 AT  %MX11732.11 : BOOL; (*RESERVED *)
	WY11708_12 AT  %MX11732.12 : BOOL; (*RESERVED *)
	WY11708_13 AT  %MX11732.13 : BOOL; (*RESERVED *)
	WY11708_14 AT  %MX11732.14 : BOOL; (*RESERVED *)
	WY11708_15 AT  %MX11732.15 : BOOL; (*RESERVED *)
	WY11708_16 AT  %MX11732.16 : BOOL; (*RESERVED *)
	WY11708_17 AT  %MX11732.17 : BOOL; (*RESERVED *)
	WY11708_18 AT  %MX11732.18 : BOOL; (*RESERVED *)
	WY11708_19 AT  %MX11732.19 : BOOL; (*RESERVED *)
	WY11708_20 AT  %MX11732.20 : BOOL; (*RESERVED *)
	WY11708_21 AT  %MX11732.21 : BOOL; (*RESERVED *)
	WY11708_22 AT  %MX11732.22 : BOOL; (*RESERVED *)
	WY11708_23 AT  %MX11732.23 : BOOL; (*RESERVED *)
	WY11708_24 AT  %MX11732.24 : BOOL; (*RESERVED *)
	WY11708_25 AT  %MX11732.25 : BOOL; (*RESERVED *)
	WY11708_26 AT  %MX11732.26 : BOOL; (*RESERVED *)
	WY11708_27 AT  %MX11732.27 : BOOL; (*RESERVED *)
	WY11708_28 AT  %MX11732.28 : BOOL; (*RESERVED *)
	WY11708_29 AT  %MX11732.29 : BOOL; (*RESERVED *)
	WY11708_30 AT  %MX11732.30 : BOOL; (*RESERVED *)
	WY11708_31 AT  %MX11732.31 : BOOL; (*RESERVED *)

	WY11709_00 AT  %MX11736.0 : BOOL; (*RESERVED *)
	WY11709_01 AT  %MX11736.1 : BOOL; (*RESERVED *)
	WY11709_02 AT  %MX11736.2 : BOOL; (*RESERVED *)
	WY11709_03 AT  %MX11736.3 : BOOL; (*RESERVED *)
	WY11709_04 AT  %MX11736.4 : BOOL; (*RESERVED *)
	WY11709_05 AT  %MX11736.5 : BOOL; (*RESERVED *)
	WY11709_06 AT  %MX11736.6 : BOOL; (*RESERVED *)
	WY11709_07 AT  %MX11736.7 : BOOL; (*RESERVED *)
	WY11709_08 AT  %MX11736.8 : BOOL; (*RESERVED *)
	WY11709_09 AT  %MX11736.9 : BOOL; (*RESERVED *)
	WY11709_10 AT  %MX11736.10 : BOOL; (*RESERVED *)
	WY11709_11 AT  %MX11736.11 : BOOL; (*RESERVED *)
	WY11709_12 AT  %MX11736.12 : BOOL; (*RESERVED *)
	WY11709_13 AT  %MX11736.13 : BOOL; (*RESERVED *)
	WY11709_14 AT  %MX11736.14 : BOOL; (*RESERVED *)
	WY11709_15 AT  %MX11736.15 : BOOL; (*RESERVED *)
	WY11709_16 AT  %MX11736.16 : BOOL; (*RESERVED *)
	WY11709_17 AT  %MX11736.17 : BOOL; (*RESERVED *)
	WY11709_18 AT  %MX11736.18 : BOOL; (*RESERVED *)
	WY11709_19 AT  %MX11736.19 : BOOL; (*RESERVED *)
	WY11709_20 AT  %MX11736.20 : BOOL; (*RESERVED *)
	WY11709_21 AT  %MX11736.21 : BOOL; (*RESERVED *)
	WY11709_22 AT  %MX11736.22 : BOOL; (*RESERVED *)
	WY11709_23 AT  %MX11736.23 : BOOL; (*RESERVED *)
	WY11709_24 AT  %MX11736.24 : BOOL; (*RESERVED *)
	WY11709_25 AT  %MX11736.25 : BOOL; (*RESERVED *)
	WY11709_26 AT  %MX11736.26 : BOOL; (*RESERVED *)
	WY11709_27 AT  %MX11736.27 : BOOL; (*RESERVED *)
	WY11709_28 AT  %MX11736.28 : BOOL; (*RESERVED *)
	WY11709_29 AT  %MX11736.29 : BOOL; (*RESERVED *)
	WY11709_30 AT  %MX11736.30 : BOOL; (*RESERVED *)
	WY11709_31 AT  %MX11736.31 : BOOL; (*RESERVED *)

	WY11710_00 AT  %MX11740.0 : BOOL; (*RESERVED *)
	WY11710_01 AT  %MX11740.1 : BOOL; (*RESERVED *)
	WY11710_02 AT  %MX11740.2 : BOOL; (*RESERVED *)
	WY11710_03 AT  %MX11740.3 : BOOL; (*RESERVED *)
	WY11710_04 AT  %MX11740.4 : BOOL; (*RESERVED *)
	WY11710_05 AT  %MX11740.5 : BOOL; (*RESERVED *)
	WY11710_06 AT  %MX11740.6 : BOOL; (*RESERVED *)
	WY11710_07 AT  %MX11740.7 : BOOL; (*RESERVED *)
	WY11710_08 AT  %MX11740.8 : BOOL; (*RESERVED *)
	WY11710_09 AT  %MX11740.9 : BOOL; (*RESERVED *)
	WY11710_10 AT  %MX11740.10 : BOOL; (*RESERVED *)
	WY11710_11 AT  %MX11740.11 : BOOL; (*RESERVED *)
	WY11710_12 AT  %MX11740.12 : BOOL; (*RESERVED *)
	WY11710_13 AT  %MX11740.13 : BOOL; (*RESERVED *)
	WY11710_14 AT  %MX11740.14 : BOOL; (*RESERVED *)
	WY11710_15 AT  %MX11740.15 : BOOL; (*RESERVED *)
	WY11710_16 AT  %MX11740.16 : BOOL; (*RESERVED *)
	WY11710_17 AT  %MX11740.17 : BOOL; (*RESERVED *)
	WY11710_18 AT  %MX11740.18 : BOOL; (*RESERVED *)
	WY11710_19 AT  %MX11740.19 : BOOL; (*RESERVED *)
	WY11710_20 AT  %MX11740.20 : BOOL; (*RESERVED *)
	WY11710_21 AT  %MX11740.21 : BOOL; (*RESERVED *)
	WY11710_22 AT  %MX11740.22 : BOOL; (*RESERVED *)
	WY11710_23 AT  %MX11740.23 : BOOL; (*RESERVED *)
	WY11710_24 AT  %MX11740.24 : BOOL; (*RESERVED *)
	WY11710_25 AT  %MX11740.25 : BOOL; (*RESERVED *)
	WY11710_26 AT  %MX11740.26 : BOOL; (*RESERVED *)
	WY11710_27 AT  %MX11740.27 : BOOL; (*RESERVED *)
	WY11710_28 AT  %MX11740.28 : BOOL; (*RESERVED *)
	WY11710_29 AT  %MX11740.29 : BOOL; (*RESERVED *)
	WY11710_30 AT  %MX11740.30 : BOOL; (*RESERVED *)
	WY11710_31 AT  %MX11740.31 : BOOL; (*RESERVED *)

	WY11711_00 AT  %MX11744.0 : BOOL; (*RESERVED *)
	WY11711_01 AT  %MX11744.1 : BOOL; (*RESERVED *)
	WY11711_02 AT  %MX11744.2 : BOOL; (*RESERVED *)
	WY11711_03 AT  %MX11744.3 : BOOL; (*RESERVED *)
	WY11711_04 AT  %MX11744.4 : BOOL; (*RESERVED *)
	WY11711_05 AT  %MX11744.5 : BOOL; (*RESERVED *)
	WY11711_06 AT  %MX11744.6 : BOOL; (*RESERVED *)
	WY11711_07 AT  %MX11744.7 : BOOL; (*RESERVED *)
	WY11711_08 AT  %MX11744.8 : BOOL; (*RESERVED *)
	WY11711_09 AT  %MX11744.9 : BOOL; (*RESERVED *)
	WY11711_10 AT  %MX11744.10 : BOOL; (*RESERVED *)
	WY11711_11 AT  %MX11744.11 : BOOL; (*RESERVED *)
	WY11711_12 AT  %MX11744.12 : BOOL; (*RESERVED *)
	WY11711_13 AT  %MX11744.13 : BOOL; (*RESERVED *)
	WY11711_14 AT  %MX11744.14 : BOOL; (*RESERVED *)
	WY11711_15 AT  %MX11744.15 : BOOL; (*RESERVED *)
	WY11711_16 AT  %MX11744.16 : BOOL; (*RESERVED *)
	WY11711_17 AT  %MX11744.17 : BOOL; (*RESERVED *)
	WY11711_18 AT  %MX11744.18 : BOOL; (*RESERVED *)
	WY11711_19 AT  %MX11744.19 : BOOL; (*RESERVED *)
	WY11711_20 AT  %MX11744.20 : BOOL; (*RESERVED *)
	WY11711_21 AT  %MX11744.21 : BOOL; (*RESERVED *)
	WY11711_22 AT  %MX11744.22 : BOOL; (*RESERVED *)
	WY11711_23 AT  %MX11744.23 : BOOL; (*RESERVED *)
	WY11711_24 AT  %MX11744.24 : BOOL; (*RESERVED *)
	WY11711_25 AT  %MX11744.25 : BOOL; (*RESERVED *)
	WY11711_26 AT  %MX11744.26 : BOOL; (*RESERVED *)
	WY11711_27 AT  %MX11744.27 : BOOL; (*RESERVED *)
	WY11711_28 AT  %MX11744.28 : BOOL; (*RESERVED *)
	WY11711_29 AT  %MX11744.29 : BOOL; (*RESERVED *)
	WY11711_30 AT  %MX11744.30 : BOOL; (*RESERVED *)
	WY11711_31 AT  %MX11744.31 : BOOL; (*RESERVED *)

	WY11712_00 AT  %MX11748.0 : BOOL; (*RESERVED *)
	WY11712_01 AT  %MX11748.1 : BOOL; (*RESERVED *)
	WY11712_02 AT  %MX11748.2 : BOOL; (*RESERVED *)
	WY11712_03 AT  %MX11748.3 : BOOL; (*RESERVED *)
	WY11712_04 AT  %MX11748.4 : BOOL; (*RESERVED *)
	WY11712_05 AT  %MX11748.5 : BOOL; (*RESERVED *)
	WY11712_06 AT  %MX11748.6 : BOOL; (*RESERVED *)
	WY11712_07 AT  %MX11748.7 : BOOL; (*RESERVED *)
	WY11712_08 AT  %MX11748.8 : BOOL; (*RESERVED *)
	WY11712_09 AT  %MX11748.9 : BOOL; (*RESERVED *)
	WY11712_10 AT  %MX11748.10 : BOOL; (*RESERVED *)
	WY11712_11 AT  %MX11748.11 : BOOL; (*RESERVED *)
	WY11712_12 AT  %MX11748.12 : BOOL; (*RESERVED *)
	WY11712_13 AT  %MX11748.13 : BOOL; (*RESERVED *)
	WY11712_14 AT  %MX11748.14 : BOOL; (*RESERVED *)
	WY11712_15 AT  %MX11748.15 : BOOL; (*RESERVED *)
	WY11712_16 AT  %MX11748.16 : BOOL; (*RESERVED *)
	WY11712_17 AT  %MX11748.17 : BOOL; (*RESERVED *)
	WY11712_18 AT  %MX11748.18 : BOOL; (*RESERVED *)
	WY11712_19 AT  %MX11748.19 : BOOL; (*RESERVED *)
	WY11712_20 AT  %MX11748.20 : BOOL; (*RESERVED *)
	WY11712_21 AT  %MX11748.21 : BOOL; (*RESERVED *)
	WY11712_22 AT  %MX11748.22 : BOOL; (*RESERVED *)
	WY11712_23 AT  %MX11748.23 : BOOL; (*RESERVED *)
	WY11712_24 AT  %MX11748.24 : BOOL; (*RESERVED *)
	WY11712_25 AT  %MX11748.25 : BOOL; (*RESERVED *)
	WY11712_26 AT  %MX11748.26 : BOOL; (*RESERVED *)
	WY11712_27 AT  %MX11748.27 : BOOL; (*RESERVED *)
	WY11712_28 AT  %MX11748.28 : BOOL; (*RESERVED *)
	WY11712_29 AT  %MX11748.29 : BOOL; (*RESERVED *)
	WY11712_30 AT  %MX11748.30 : BOOL; (*RESERVED *)
	WY11712_31 AT  %MX11748.31 : BOOL; (*RESERVED *)

	WY11713_00 AT  %MX11752.0 : BOOL; (*RESERVED *)
	WY11713_01 AT  %MX11752.1 : BOOL; (*RESERVED *)
	WY11713_02 AT  %MX11752.2 : BOOL; (*RESERVED *)
	WY11713_03 AT  %MX11752.3 : BOOL; (*RESERVED *)
	WY11713_04 AT  %MX11752.4 : BOOL; (*RESERVED *)
	WY11713_05 AT  %MX11752.5 : BOOL; (*RESERVED *)
	WY11713_06 AT  %MX11752.6 : BOOL; (*RESERVED *)
	WY11713_07 AT  %MX11752.7 : BOOL; (*RESERVED *)
	WY11713_08 AT  %MX11752.8 : BOOL; (*RESERVED *)
	WY11713_09 AT  %MX11752.9 : BOOL; (*RESERVED *)
	WY11713_10 AT  %MX11752.10 : BOOL; (*RESERVED *)
	WY11713_11 AT  %MX11752.11 : BOOL; (*RESERVED *)
	WY11713_12 AT  %MX11752.12 : BOOL; (*RESERVED *)
	WY11713_13 AT  %MX11752.13 : BOOL; (*RESERVED *)
	WY11713_14 AT  %MX11752.14 : BOOL; (*RESERVED *)
	WY11713_15 AT  %MX11752.15 : BOOL; (*RESERVED *)
	WY11713_16 AT  %MX11752.16 : BOOL; (*RESERVED *)
	WY11713_17 AT  %MX11752.17 : BOOL; (*RESERVED *)
	WY11713_18 AT  %MX11752.18 : BOOL; (*RESERVED *)
	WY11713_19 AT  %MX11752.19 : BOOL; (*RESERVED *)
	WY11713_20 AT  %MX11752.20 : BOOL; (*RESERVED *)
	WY11713_21 AT  %MX11752.21 : BOOL; (*RESERVED *)
	WY11713_22 AT  %MX11752.22 : BOOL; (*RESERVED *)
	WY11713_23 AT  %MX11752.23 : BOOL; (*RESERVED *)
	WY11713_24 AT  %MX11752.24 : BOOL; (*RESERVED *)
	WY11713_25 AT  %MX11752.25 : BOOL; (*RESERVED *)
	WY11713_26 AT  %MX11752.26 : BOOL; (*RESERVED *)
	WY11713_27 AT  %MX11752.27 : BOOL; (*RESERVED *)
	WY11713_28 AT  %MX11752.28 : BOOL; (*RESERVED *)
	WY11713_29 AT  %MX11752.29 : BOOL; (*RESERVED *)
	WY11713_30 AT  %MX11752.30 : BOOL; (*RESERVED *)
	WY11713_31 AT  %MX11752.31 : BOOL; (*RESERVED *)

	WY11714_00 AT  %MX11756.0 : BOOL; (*RESERVED *)
	WY11714_01 AT  %MX11756.1 : BOOL; (*RESERVED *)
	WY11714_02 AT  %MX11756.2 : BOOL; (*RESERVED *)
	WY11714_03 AT  %MX11756.3 : BOOL; (*RESERVED *)
	WY11714_04 AT  %MX11756.4 : BOOL; (*RESERVED *)
	WY11714_05 AT  %MX11756.5 : BOOL; (*RESERVED *)
	WY11714_06 AT  %MX11756.6 : BOOL; (*RESERVED *)
	WY11714_07 AT  %MX11756.7 : BOOL; (*RESERVED *)
	WY11714_08 AT  %MX11756.8 : BOOL; (*RESERVED *)
	WY11714_09 AT  %MX11756.9 : BOOL; (*RESERVED *)
	WY11714_10 AT  %MX11756.10 : BOOL; (*RESERVED *)
	WY11714_11 AT  %MX11756.11 : BOOL; (*RESERVED *)
	WY11714_12 AT  %MX11756.12 : BOOL; (*RESERVED *)
	WY11714_13 AT  %MX11756.13 : BOOL; (*RESERVED *)
	WY11714_14 AT  %MX11756.14 : BOOL; (*RESERVED *)
	WY11714_15 AT  %MX11756.15 : BOOL; (*RESERVED *)
	WY11714_16 AT  %MX11756.16 : BOOL; (*RESERVED *)
	WY11714_17 AT  %MX11756.17 : BOOL; (*RESERVED *)
	WY11714_18 AT  %MX11756.18 : BOOL; (*RESERVED *)
	WY11714_19 AT  %MX11756.19 : BOOL; (*RESERVED *)
	WY11714_20 AT  %MX11756.20 : BOOL; (*RESERVED *)
	WY11714_21 AT  %MX11756.21 : BOOL; (*RESERVED *)
	WY11714_22 AT  %MX11756.22 : BOOL; (*RESERVED *)
	WY11714_23 AT  %MX11756.23 : BOOL; (*RESERVED *)
	WY11714_24 AT  %MX11756.24 : BOOL; (*RESERVED *)
	WY11714_25 AT  %MX11756.25 : BOOL; (*RESERVED *)
	WY11714_26 AT  %MX11756.26 : BOOL; (*RESERVED *)
	WY11714_27 AT  %MX11756.27 : BOOL; (*RESERVED *)
	WY11714_28 AT  %MX11756.28 : BOOL; (*RESERVED *)
	WY11714_29 AT  %MX11756.29 : BOOL; (*RESERVED *)
	WY11714_30 AT  %MX11756.30 : BOOL; (*RESERVED *)
	WY11714_31 AT  %MX11756.31 : BOOL; (*RESERVED *)

	WY11715_00 AT  %MX11760.0 : BOOL; (*RESERVED *)
	WY11715_01 AT  %MX11760.1 : BOOL; (*RESERVED *)
	WY11715_02 AT  %MX11760.2 : BOOL; (*RESERVED *)
	WY11715_03 AT  %MX11760.3 : BOOL; (*RESERVED *)
	WY11715_04 AT  %MX11760.4 : BOOL; (*RESERVED *)
	WY11715_05 AT  %MX11760.5 : BOOL; (*RESERVED *)
	WY11715_06 AT  %MX11760.6 : BOOL; (*RESERVED *)
	WY11715_07 AT  %MX11760.7 : BOOL; (*RESERVED *)
	WY11715_08 AT  %MX11760.8 : BOOL; (*RESERVED *)
	WY11715_09 AT  %MX11760.9 : BOOL; (*RESERVED *)
	WY11715_10 AT  %MX11760.10 : BOOL; (*RESERVED *)
	WY11715_11 AT  %MX11760.11 : BOOL; (*RESERVED *)
	WY11715_12 AT  %MX11760.12 : BOOL; (*RESERVED *)
	WY11715_13 AT  %MX11760.13 : BOOL; (*RESERVED *)
	WY11715_14 AT  %MX11760.14 : BOOL; (*RESERVED *)
	WY11715_15 AT  %MX11760.15 : BOOL; (*RESERVED *)
	WY11715_16 AT  %MX11760.16 : BOOL; (*RESERVED *)
	WY11715_17 AT  %MX11760.17 : BOOL; (*RESERVED *)
	WY11715_18 AT  %MX11760.18 : BOOL; (*RESERVED *)
	WY11715_19 AT  %MX11760.19 : BOOL; (*RESERVED *)
	WY11715_20 AT  %MX11760.20 : BOOL; (*RESERVED *)
	WY11715_21 AT  %MX11760.21 : BOOL; (*RESERVED *)
	WY11715_22 AT  %MX11760.22 : BOOL; (*RESERVED *)
	WY11715_23 AT  %MX11760.23 : BOOL; (*RESERVED *)
	WY11715_24 AT  %MX11760.24 : BOOL; (*RESERVED *)
	WY11715_25 AT  %MX11760.25 : BOOL; (*RESERVED *)
	WY11715_26 AT  %MX11760.26 : BOOL; (*RESERVED *)
	WY11715_27 AT  %MX11760.27 : BOOL; (*RESERVED *)
	WY11715_28 AT  %MX11760.28 : BOOL; (*RESERVED *)
	WY11715_29 AT  %MX11760.29 : BOOL; (*RESERVED *)
	WY11715_30 AT  %MX11760.30 : BOOL; (*RESERVED *)
	WY11715_31 AT  %MX11760.31 : BOOL; (*RESERVED *)

END_VAR

// ---- GVLs/Digital_Ctrl/Global_Variables_DigitalMapping.TcGVL
{attribute 'Tc2GvlVarNames'}
VAR_GLOBAL

(* xxxxxxxxxxxxxxxxxxxxxxxxxxxxxxxx DIGITAL INPUT xxxxxxxxxxxxxxxxxxxxxxxxxxxxxxxx*)
(*========================================================================*)
(*
	X100_00  AT %I* : BOOL; (*GENERAL ALARM PB - RESET (-100S1)*)
	X100_01  AT %I* : BOOL; (*GENERAL BUZZER PB - RESET (-100S2)*)
	X100_02  AT %I* : BOOL; (*GENERAL MAIN PANEL PB - E-STOP (-100S3)*)
	X100_03  AT %I* : BOOL; (*OPERATOR PULL STRING - E-STOP (-100S4)*)
	X100_04  AT %I* : BOOL; (*MAINTENANCE E/STOP PULL STRING (-100S5)*)
	X100_05  AT %I* : BOOL; (*GENERAL PHASE SEQEUNCE RELAY - TRIP (-8K1)*)
	X100_06  AT %I* : BOOL; (*STN 1 PROCESS TANK PUMP TOR - TRIP (-50F2)*)
	X100_07  AT %I* : BOOL; (*STN 2 PROCESS TANK PUMP TOR - TRIP (-51F2)*)
	X100_08  AT %I* : BOOL; (*STN 3 PROCESS TANK PUMP TOR - TRIP (-52F2)*)
	X100_09  AT %I* : BOOL; (*STN 2&3 AGITATION MOTOR TOR - TRIP (-25F2)*)
	X100_10  AT %I* : BOOL; (*STN 5 BLOWER TOR - TRIP (-65F2)*)
	X100_11  AT %I* : BOOL; (*STN 5 VACUUM PUMP TOR - TRIP (-56F2)*)
	X100_12  AT %I* : BOOL; (*RESERVED*)
	X100_13  AT %I* : BOOL; (*RESERVED*)
	X100_14  AT %I* : BOOL; (*RESERVED*)
	X100_15  AT %I* : BOOL; (*RESERVED*)

	X101_00  AT %I* : BOOL; (*STN 1 SLIDING DOOR RS - OPEN (-101S5)*)
	X101_01  AT %I* : BOOL; (*STN 1 SLIDING DOOR RS - CLOSE (-101S6)*)
	X101_02  AT %I* : BOOL; (*ARM 1 HORZ SENSOR - LD SIDE OT  (-101B1)*)
	X101_03  AT %I* : BOOL; (*ARM 1 HORZ SENSOR - HOME (-101B2)*)
	X101_04  AT %I* : BOOL; (*STN 1 SUB PROCESS TANK HEATER THERMOSTAT A - ALARM (-101S8)*)
	X101_05  AT %I* : BOOL; (*STN 1 SUB PROCESS TANK HEATER THERMOSTAT B - ALARM (-101S9)*)
	X101_06  AT %I* : BOOL; (*STN 1 PROCESS TANK SENSOR - MIN LEVEL (-101S1)*)
	X101_07  AT %I* : BOOL; (*STN 1 SUB PROCESS TANK SENSOR - REG LEVEL (-101S2)*)
	X101_08  AT %I* : BOOL; (*STN 1 SUB PROCESS TANK SENSOR - MIN LEVEL (-101S3)*)
	X101_09  AT %I* : BOOL; (*DETERGENT STORAGE TANK SENSOR - MIN LEVEL (-101S4)*)
	X101_10  AT %I* : BOOL; (*STRUCTURE 1 DRIP PAN SENSOR - LEAK (-101B3)*)
	X101_11  AT %I* : BOOL; (*STN 1 SUB PROCESS TANK SENSOR - TOP UP LEVEL (-101S7)*)
	X101_12  AT %I* : BOOL; (*RESERVED*)
	X101_13  AT %I* : BOOL; (*RESERVED*)
	X101_14  AT %I* : BOOL; (*RESERVED*)
	X101_15  AT %I* : BOOL; (*RESERVED*)

	X102_00  AT %I* : BOOL; (*MODULE 1 DOOR MAGNETIC SWITCH FRONT MAINTENANCE TOP - ALARM (-102S1,2,3)*)
	X102_01  AT %I* : BOOL; (*RESERVED*)
	X102_02  AT %I* : BOOL; (*RESERVED*)
	X102_03  AT %I* : BOOL; (*MODULE 1 SLIDING DOOR SENSOR A (-102B7)*)
	X102_04  AT %I* : BOOL; (*MODULE 1 SLIDING DOOR SENSOR B (-102B8)*)
	X102_05  AT %I* : BOOL; (*RESERVED*)
	X102_06  AT %I* : BOOL; (*RESERVED*)
	X102_07  AT %I* : BOOL; (*RESERVED*)
	X102_08  AT %I* : BOOL; (*RESERVED*)
	X102_09  AT %I* : BOOL; (*RESERVED*)
	X102_10  AT %I* : BOOL; (*RESERVED*)
	X102_11  AT %I* : BOOL; (*RESERVED*)
	X102_12  AT %I* : BOOL; (*RESERVED*)
	X102_13  AT %I* : BOOL; (*RESERVED*)
	X102_14  AT %I* : BOOL; (*RESERVED*)
	X102_15  AT %I* : BOOL; (*RESERVED*)

	X110_00  AT %I* : BOOL; (*STN 2 PROCESS TANK SENSOR - MIN LEVEL (-110S1)*)
	X110_01  AT %I* : BOOL; (*STN 2 SUB PROCESS TANK SENSOR - REG LEVEL (-110S2)*)
	X110_02  AT %I* : BOOL; (*STN 2 SUB PROCESS TANK SENSOR - MIN LEVEL (-110S3)*)
	X110_03  AT %I* : BOOL; (*STN 3 PROCESS TANK SENSOR - MIN LEVEL (-110S4)*)
	X110_04  AT %I* : BOOL; (*STN 3 SUB PROCESS TANK SENSOR - REG LEVEL (-110S5)*)
	X110_05  AT %I* : BOOL; (*STN 3 SUB PROCESS TANK SENSOR - MIN LEVEL (-110S6)*)
	X110_06  AT %I* : BOOL; (*ARM 1 VERT SENSOR - TOP SIDE OT (-110B1)*)
	X110_07  AT %I* : BOOL; (*ARM 1 VERT SENSOR - TOP SIDE HOME (-110B2)*)
	X110_08  AT %I* : BOOL; (*ARM 1 VERT SENSOR - BOTTOM SIDE OT (-110B3)*)
	X110_09  AT %I* : BOOL; (*ARM 1 VERT SENSOR - CRASH (-110B4)*)
	X110_10  AT %I* : BOOL; (*ARM 1 SENSOR A - MISSHOOK (-110B5)*)
	X110_11  AT %I* : BOOL; (*ARM 1 SENSOR B - MISSHOOK (-110B6)*)
	X110_12  AT %I* : BOOL; (*RESERVED*)
	X110_13  AT %I* : BOOL; (*RESERVED*)
	X110_14  AT %I* : BOOL; (*RESERVED*)
	X110_15  AT %I* : BOOL; (*RESERVED*)

	X111_00  AT %I* : BOOL; (*STRUCTURE 2 DRIP PAN SENSOR - LEAK (-111B1)*)
	X111_01  AT %I* : BOOL; (*STN 2 SUB PROCESS TANK HEATER THERMOSTAT A - ALARM (-111S1)*)
	X111_02  AT %I* : BOOL; (*STN 2 SUB PROCESS TANK HEATER THERMOSTAT B - ALARM (-111S2)*)
	X111_03  AT %I* : BOOL; (*STN 3 SUB PROCESS TANK HEATER THERMOSTAT A - ALARM (-111S3)*)
	X111_04  AT %I* : BOOL; (*STN 3 SUB PROCESS TANK HEATER THERMOSTAT B - ALARM (-111S4)*)
	X111_05  AT %I* : BOOL; (*MODULE 2 DOOR MAGNETIC SWITCH FRONT MAINTENANCE TOP - ALARM (-111S11,12)*)
	X111_06  AT %I* : BOOL; (*RESERVED*)
	X111_07  AT %I* : BOOL; (*RESERVED*)
	X111_08  AT %I* : BOOL; (*MODULE 2 SLIDING DOOR SENSOR A (-111B2)*)
	X111_09  AT %I* : BOOL; (*MODULE 2 SLIDING DOOR SENSOR B (-111B3)*)
	X111_10  AT %I* : BOOL; (*MODULE 2 SLIDING DOOR SENSOR C (-111B4)*)
	X111_11  AT %I* : BOOL; (*RESERVED*)
	X111_12  AT %I* : BOOL; (*RESERVED*)
	X111_13  AT %I* : BOOL; (*RESERVED*)
	X111_14  AT %I* : BOOL; (*RESERVED*)
	X111_15  AT %I* : BOOL; (*RESERVED*)

	X115_00  AT %I* : BOOL; (*ARM 1 HORZ SENSOR - ULD SIDE OT (-115B1)*)
	X115_01  AT %I* : BOOL; (*ULD CONVEYOR SENSOR - FEED (-115B2)*)
	X115_02  AT %I* : BOOL; (*ULD CONVEYOR SENSOR - PICK (-115B3)*)
	X115_03  AT %I* : BOOL; (*ULD CONVEYOR PB - RAPID (-115S11)*)
	X115_04  AT %I* : BOOL; (*ULD CONVEYOR PB - E-STOP (-115S12)*)
	X115_05  AT %I* : BOOL; (*STN 4 SLIDING DOOR RS - OPEN (-115S1)*)
	X115_06  AT %I* : BOOL; (*STN 4 SLIDING DOOR RS - CLOSE (-115S2)*)
	X115_07  AT %I* : BOOL; (*STN 5 SLIDING DOOR RS - OPEN (-115S3)*)
	X115_08  AT %I* : BOOL; (*STN 5 SLIDING DOOR RS - CLOSE (-115S4)*)
	X115_09  AT %I* : BOOL; (*STN 5 SLIDING DOOR RS_A - CLAMP (-115S5)*)
	X115_10  AT %I* : BOOL; (*STN 5 SLIDING DOOR RS_A - UNCLAMP (-115S6)*)
	X115_11  AT %I* : BOOL; (*STN 5 SLIDING DOOR RS_B - CLAMP (-115S7)*)
	X115_12  AT %I* : BOOL; (*STN 5 SLIDING DOOR RS_B - UNCLAMP (-115S8)*)
	X115_13  AT %I* : BOOL; (*STN 5 PROCESS TANK HEATER THERMOSTAT - ALARM (-115S9)*)
	X115_14  AT %I* : BOOL; (*GENERAL INCOMING FLOW SENSOR - MIN FLOW (-115B4)*)
	X115_15  AT %I* : BOOL; (*RESERVED*)

	X116_00  AT %I* : BOOL; (*MAIN INC HEATER THERMOSTAT A - ALARM (-116S1)*)
	X116_01  AT %I* : BOOL; (*MAIN INC HEATER THERMOSTAT B - ALARM (-116S2)*)
	X116_02  AT %I* : BOOL; (*STN 4 IONIZER ION LEVEL ALARM (-116U1)*)
	X116_03  AT %I* : BOOL; (*STN 4 IONIZER CONDITION ALARM (-116U1)*)
	X116_04  AT %I* : BOOL; (*STN 4 IONIZER ALARM OUTPUT (-116U1)*)
	X116_05  AT %I* : BOOL; (*UNLOADING IONIZER ION LEVEL ALARM (-116U2)*)
	X116_06  AT %I* : BOOL; (*UNLOADING IONIZER CONDITION ALARM (-116U2)*)
	X116_07  AT %I* : BOOL; (*UNLOADING IONIZER ALARM OUTPUT (-116U2)*)
	X116_08  AT %I* : BOOL; (*MODULE 3 DOOR MAGNETIC SWITCH FRONT MAINTENANCE TOP - ALARM (-116S3,4,5,6,7,8,9)*)
	X116_09  AT %I* : BOOL; (*RESERVED*)
	X116_10  AT %I* : BOOL; (*RESERVED*)
	X116_11  AT %I* : BOOL; (*MODULE 3 SLIDING DOOR SENSOR A (-116B1)*)
	X116_12  AT %I* : BOOL; (*MODULE 3 SLIDING DOOR SENSOR B (-116B2)*)
	X116_13  AT %I* : BOOL; (*MODULE 3 SLIDING DOOR SENSOR C (-116B3)*)
	X116_14  AT %I* : BOOL; (*RESERVED*)
	X116_15  AT %I* : BOOL; (*RESERVED*)

	X117_00  AT %I* : BOOL; (*ULD CYLINDER - UP SENSOR A (-117S1)*)
	X117_01  AT %I* : BOOL; (*ULD CYLINDER - DOWN SENSOR A (-117S2)*)
	X117_02  AT %I* : BOOL; (*ULD CYLINDER - UP SENSOR B (-117S3)*)
	X117_03  AT %I* : BOOL; (*ULD CYLINDER - DOWN SENSOR B (-117S4)*)
	X117_04  AT %I* : BOOL; (*ULD CYLINDER - FORWARD SENSOR (-117S5)*)
	X117_05  AT %I* : BOOL; (*ULD CYLINDER - REVERSE SENSOR (-117S6)*)
	X117_06  AT %I* : BOOL; (*STN 4 CDA CYLINDER - IN (-117S7)*)
	X117_07  AT %I* : BOOL; (*STN 4 CDA CYLINDER - OUT (-117S8)*)
	X117_08  AT %I* : BOOL; (*RESERVED*)
	X117_09  AT %I* : BOOL; (*RESERVED*)
	X117_10  AT %I* : BOOL; (*RESERVED*)
	X117_11  AT %I* : BOOL; (*RESERVED*)
	X117_12  AT %I* : BOOL; (*RESERVED*)
	X117_13  AT %I* : BOOL; (*RESERVED*)
	X117_14  AT %I* : BOOL; (*RESERVED*)
	X117_15  AT %I* : BOOL; (*RESERVED*)

	X120_00  AT %I* : BOOL; (*LD CONVEYOR SENSOR - FEED (-120B1)*)
	X120_01  AT %I* : BOOL; (*LD CONVEYOR SENSOR - PICK (-120B2)*)
	X120_02  AT %I* : BOOL; (*LD CONVEYOR PB - RAPID (-120S1)*)
	X120_03  AT %I* : BOOL; (*LD CONVEYOR PB - E-STOP (-120S2)*)
	X120_04  AT %I* : BOOL; (*LD CYLINDER - UP SENSOR A ()*)
	X120_05  AT %I* : BOOL; (*LD CYLINDER - DOWN SENSOR A ()*)
	X120_06  AT %I* : BOOL; (*LD CYLINDER - UP SENSOR B ()*)
	X120_07  AT %I* : BOOL; (*LD CYLINDER - DOWN SENSOR B ()*)
	X120_08  AT %I* : BOOL; (*LD CYLINDER - FORWARD SENSOR ()*)
	X120_09  AT %I* : BOOL; (*LD CYLINDER - REVERSE SENSOR ()*)
	X120_10  AT %I* : BOOL; (*RESERVED*)
	X120_11  AT %I* : BOOL; (*RESERVED*)
	X120_12  AT %I* : BOOL; (*RESERVED*)
	X120_13  AT %I* : BOOL; (*RESERVED*)
	X120_14  AT %I* : BOOL; (*RESERVED*)
	X120_15  AT %I* : BOOL; (*RESERVED*)

(* xxxxxxxxxxxxxxxxxxxxxxxxxxxxxxxx DIGITAL OUTPUT xxxxxxxxxxxxxxxxxxxxxxxxxxxxxxxx*)
(*========================================================================*)

	Y100_00  AT %Q* : BOOL; (*GENERAL ALARM RESET IND (-100S1)*)
	Y100_01  AT %Q* : BOOL; (*GENERAL BUZZER RESET IND (-100S2)*)
	Y100_02  AT %Q* : BOOL; (*GENERAL BUZZER TONE 1 (-150H3)*)
	Y100_03  AT %Q* : BOOL; (*GENERAL BUZZER TONE 2 (-150H3)*)
	Y100_04  AT %Q* : BOOL; (*GENERAL TOWER LIGHT IND - RED (-150H5)*)
	Y100_05  AT %Q* : BOOL; (*GENERAL TOWER LIGHT IND - YELLOW (-150H5)*)
	Y100_06  AT %Q* : BOOL; (*GENERAL TOWER LIGHT IND - GREEN (-150H5)*)
	Y100_07  AT %Q* : BOOL; (*RESERVED*)
	Y100_08  AT %Q* : BOOL; (*RESERVED*)
	Y100_09  AT %Q* : BOOL; (*RESERVED*)
	Y100_10  AT %Q* : BOOL; (*RESERVED*)
	Y100_11  AT %Q* : BOOL; (*RESERVED*)
	Y100_12  AT %Q* : BOOL; (*RESERVED*)
	Y100_13  AT %Q* : BOOL; (*RESERVED*)
	Y100_14  AT %Q* : BOOL; (*RESERVED*)
	Y100_15  AT %Q* : BOOL; (*RESERVED*)

	Y101_00  AT %Q* : BOOL; (*STN 1 PROCESS TANK PUMP ON/OFF (-50K1)*)
	Y101_01  AT %Q* : BOOL; (*STN 2 PROCESS TANK PUMP ON/OFF (-51K1)*)
	Y101_02  AT %Q* : BOOL; (*STN 3 PROCESS TANK PUMP ON/OFF (-52K1)*)
	Y101_03  AT %Q* : BOOL; (*STN 5 VACUUM PUMP ON/OFF (-56K1)*)
	Y101_04  AT %Q* : BOOL; (*STN 2&3 AGITATION MOTOR ON/OFF (-25K1)*)
	Y101_05  AT %Q* : BOOL; (*STN 5 BLOWER ON/OFF (-65K1)*)
	Y101_06  AT %Q* : BOOL; (*STN 1 SUB PROCESS TANK STIRRING MOTOR ON/OFF (-26K1)*)
	Y101_07  AT %Q* : BOOL; (*DETERGENT TANK 1 STIRRING MOTOR ON/OFF (-27K1)*)
	Y101_08  AT %Q* : BOOL; (*STN 1 ULTRASONIC ON/OFF (-16K1)*)
	Y101_09  AT %Q* : BOOL; (*STN 2 ULTRASONIC ON/OFF (-17K1)*)
	Y101_10  AT %Q* : BOOL; (*STN 3 ULTRASONIC ON/OFF (-18K1)*)
	Y101_11  AT %Q* : BOOL; (*STN 1 ELECTRIC ACTUATOR ON/OFF (-21K1)*)
	Y101_12  AT %Q* : BOOL; (*STN 2 ELECTRIC ACTUATOR ON/OFF (-22K1)*)
	Y101_13  AT %Q* : BOOL; (*STN 3 ELECTRIC ACTUATOR ON/OFF (-23K1)*)
	Y101_14  AT %Q* : BOOL; (*RESERVED*)
	Y101_15  AT %Q* : BOOL; (*RESERVED*)

	Y102_00  AT %Q* : BOOL; (*STN 5 PROCESS TANK HEATER A ON/OFF (-70K1)*)
	Y102_01  AT %Q* : BOOL; (*STN 5 PROCESS TANK HEATER B ON/OFF (-71K1)*)
	Y102_02  AT %Q* : BOOL; (*STN 1 SUB PROCESS TANK HEATER ON/OFF (-72K1)*)
	Y102_03  AT %Q* : BOOL; (*STN 2 SUB PROCESS TANK HEATER ON/OFF (-73K1)*)
	Y102_04  AT %Q* : BOOL; (*STN 3 SUB PROCESS TANK HEATER ON/OFF (-74K1)*)
	Y102_05  AT %Q* : BOOL; (*MAIN INC HEATER ON/OFF   (-75K1)*)
	Y102_06  AT %Q* : BOOL; (*STN 1 ULTRASONIC FREQ ON/OFF (-16U1)*)
	Y102_07  AT %Q* : BOOL; (*STN 2 ULTRASONIC FREQ ON/OFF (-17U1)*)
	Y102_08  AT %Q* : BOOL; (*STN 3 ULTRASONIC FREQ ON/OFF (-18U1)*)
	Y102_09  AT %Q* : BOOL; (*RESERVED*)
	Y102_10  AT %Q* : BOOL; (*RESERVED*)
	Y102_11  AT %Q* : BOOL; (*RESERVED*)
	Y102_12  AT %Q* : BOOL; (*RESERVED*)
	Y102_13  AT %Q* : BOOL; (*RESERVED*)
	Y102_14  AT %Q* : BOOL; (*RESERVED*)
	Y102_15  AT %Q* : BOOL; (*RESERVED*)

	Y115_00  AT %Q* : BOOL; (*STN 1 SLIDING DOOR - OPEN (-160Y1)*)
	Y115_01  AT %Q* : BOOL; (*STN 1 SLIDING DOOR - CLOSE (-160Y2)*)
	Y115_02  AT %Q* : BOOL; (*STN 4 SLIDING DOOR - OPEN (-160Y3)*)
	Y115_03  AT %Q* : BOOL; (*STN 4 SLIDING DOOR - CLOSE (-160Y4)*)
	Y115_04  AT %Q* : BOOL; (*STN 5 SLIDING DOOR - OPEN (-160Y5)*)
	Y115_05  AT %Q* : BOOL; (*STN 5 SLIDING DOOR - CLOSE (-160Y6)*)
	Y115_06  AT %Q* : BOOL; (*STN 5 SLIDING DOOR - CLAMP (-160Y7)*)
	Y115_07  AT %Q* : BOOL; (*STN 5 SLIDING DOOR - UNCLAMP (-160Y8)*)
	Y115_08  AT %Q* : BOOL; (*LD CYLINDER - UP (-160Y9)*)
	Y115_09  AT %Q* : BOOL; (*LD CYLINDER - DOWN (-160Y10)*)
	Y115_10  AT %Q* : BOOL; (*LD CYLINDER - FRONT (-160Y11)*)
	Y115_11  AT %Q* : BOOL; (*LD CYLINDER - BACK (-160Y12)*)
	Y115_12  AT %Q* : BOOL; (*ULD CYLINDER - UP (-160Y13)*)
	Y115_13  AT %Q* : BOOL; (*ULD CYLINDER - DOWN (-160Y14)*)
	Y115_14  AT %Q* : BOOL; (*ULD CYLINDER - FRONT (-160Y15)*)
	Y115_15  AT %Q* : BOOL; (*ULD CYLINDER - BACK (-160Y16)*)

	Y116_00  AT %Q* : BOOL; (*GENERAL INCOMING DIW SUPPLY AVINC-1 (-161Y1)*)
	Y116_01  AT %Q* : BOOL; (*STN 1 PROCESS TANK INCOMING DI SUPPLY AV1-1 (-161Y2)*)
	Y116_02  AT %Q* : BOOL; (*STN 1 SUB TANK INCOMING DIW SUPPLY AV1-2 (-161Y3)*)
	Y116_03  AT %Q* : BOOL; (*STN 1 DETERGENT SUPPLY 3-2 WAY AV1-3 (-161Y4)*)
	Y116_04  AT %Q* : BOOL; (*STN 2 PROCESS TANK INCOMING DIW SUPPLY AV2-1 (-161Y5)*)
	Y116_05  AT %Q* : BOOL; (*STN 3 PROCESS TANK INCOMING DIW SUPPLY AV3-1 (-161Y6)*)
	Y116_06  AT %Q* : BOOL; (*STN 4 PROCESS TANK CDA DISCHARGE AV4-1 (-161Y7)*)
	Y116_07  AT %Q* : BOOL; (*STN 4 PROCESS TANK CDA DISCHARGE AV4-2 (-161Y8)*)
	Y116_08  AT %Q* : BOOL; (*STN 5 PROCESS TANK VACUUM SUCTION AV5-1 (-161Y9)*)
	Y116_09  AT %Q* : BOOL; (*STN 5 PROCESS TANK VACUUM RELEASE AV5-2 (-161Y10)*)
	Y116_10  AT %Q* : BOOL; (*STN 5 BLOWER PROTECTION BUTTLEFLY AV5-3 (-161Y11)*)
	Y116_11  AT %Q* : BOOL; (*STN 5 BLOWER PROTECTION BUTTLEFLY AV5-4 (-161Y12)*)
	Y116_12  AT %Q* : BOOL; (*FACILITY CHILL WATER SUPPLY AV5-5 (-161Y13)*)
	Y116_13  AT %Q* : BOOL; (*STN 4 & UNLOADING IONIZER CDA DISCHARGE AVION-1 (-161Y14,15)*)
	Y116_14  AT %Q* : BOOL; (*STN 4 IONIZER STATIC ELIMINATION STOP SIGNAL (-161U1)*)
	Y116_15  AT %Q* : BOOL; (*UNLOADING IONIZER STATIC ELIMINATION STOP SIGNAL (-161U2)*)

	Y117_00  AT %Q* : BOOL; (*STN 4 CDA CYLINDER - IN (-162Y1)*)
	Y117_01  AT %Q* : BOOL; (*STN 4 CDA CYLINDER - OUT (-162Y2)*)
	Y117_02  AT %Q* : BOOL; (*RAMP PUMP AV (-162Y3)*)
	Y117_03  AT %Q* : BOOL; (*RESERVED*)
	Y117_04  AT %Q* : BOOL; (*RESERVED*)
	Y117_05  AT %Q* : BOOL; (*RESERVED*)
	Y117_06  AT %Q* : BOOL; (*RESERVED*)
	Y117_07  AT %Q* : BOOL; (*RESERVED*)
	Y117_08  AT %Q* : BOOL; (*RESERVED*)
	Y117_09  AT %Q* : BOOL; (*RESERVED*)
	Y117_10  AT %Q* : BOOL; (*RESERVED*)
	Y117_11  AT %Q* : BOOL; (*RESERVED*)
	Y117_12  AT %Q* : BOOL; (*RESERVED*)
	Y117_13  AT %Q* : BOOL; (*RESERVED*)
	Y117_14  AT %Q* : BOOL; (*RESERVED*)
	Y117_15  AT %Q* : BOOL; (*RESERVED*)
*)
END_VAR

// ---- GVLs/Digital_Ctrl/Global_Variables_Digital_Persistent.TcGVL
{attribute 'Tc2GvlVarNames'}
VAR_GLOBAL PERSISTENT

(* xxxxxxxxxxxxxxxxxxxxxxxxxxxxxxxx DEACTIVATED xxxxxxxxxxxxxxxxxxxxxxxxxxxxxxxx*)
(*========================================================================*)


	ARbArmMissHookByPass1				: ARRAY [1..iArmQty] OF BOOL;
	ARbArmMissHookByPass2				: ARRAY [1..iArmQty] OF BOOL;
	ARbArmCrashByPass					: ARRAY [1..iArmQty] OF BOOL;
	ARbConductivityBypass				: ARRAY [1..iStnQty] OF BOOL;
	ARbResistivityBypass					: ARRAY [1..iStnQty] OF BOOL;
	bIncResistivityBypass					: BOOL;
	ARbFilterPressureBypass				: ARRAY [1..iStnQty] OF BOOL;
	ARbFlowSwitchBypass					: ARRAY [1..iStnQty] OF BOOL;
	ARbIncFlowSwitchBypass				: ARRAY [1..iStnQty] OF BOOL;
	ARbPhBypass						: ARRAY [1..iStnQty] OF BOOL;
	bSafetyDoorSensorBypass				: BOOL;
	bStandaloneInlineHeaterBypass			: BOOL;

	ARlrArmDetectZoneRange				: ARRAY [1..iStnQty] OF LREAL;
	ARlrArmStnDetectZoneRange			: ARRAY [1..iArmQty,1..iStnQty] OF LREAL;
	ARiArmDeactDetectZoneRange			: ARRAY [1..iArmQty] OF INT;
	ARbArmMisshook1Alarm				: ARRAY [1..iArmQty] OF BOOL;
	ARbArmMisshook2Alarm				: ARRAY [1..iArmQty] OF BOOL;

	ARbStationFunctionBypass				: ARRAY [1..iStnQty] OF BOOL;

	bStnLiftoutMechanismBypass			: BOOL;

	bBuzzerDisable						: BOOL;
	bUnloadingBuzzerDisable				: BOOL;

	ARbMultiStnAgitationBypass			: ARRAY [1..iStnQty] OF BOOL;

END_VAR

// ---- GVLs/General_Ctrl/Global_Variables.TcGVL
{attribute 'Tc2GvlVarNames'}
VAR_GLOBAL

(* xxxxxxxxxxxxxxxxxxxxxxx Conveyor Motor R_TRIG and F_TRIG xxxxxxxxxxxxxxxxxxxxxxx*)
(*========================================================================*)

	bBasketCfmEn										: BOOL;
	ARbBasketGdFlag									: ARRAY [0..20] OF BOOL;
	ARbBasketBdFlag									: ARRAY [0..20] OF BOOL;

	bLdConveyorMotorOnOffAbnormalFlag					: BOOL;
	bUldConveyorMotorOnOffAbnormalFlag					: BOOL;

	bStn9BasketNextTransferAvailableFlag					: BOOL;
	bStn10BasketNextTransferAvailableFlag					: BOOL;

	bMotorRotateHoming 									: BOOL;

	LdMotor1RE											: R_TRIG;
	LdMotor1FE											: F_TRIG;
	LdMotor2RE											: R_TRIG;
	LdMotor2FE											: F_TRIG;
	LdMotor3RE											: R_TRIG;
	LdMotor3FE											: F_TRIG;
	LdMotor4RE											: R_TRIG;
	LdMotor4FE											: F_TRIG;
	LdMotor5RE											: R_TRIG;
	LdMotor5FE											: F_TRIG;

	UldMotor1RE											: R_TRIG;
	UldMotor1FE											: F_TRIG;
	UldMotor2RE											: R_TRIG;
	UldMotor2FE											: F_TRIG;
	UldMotor3RE											: R_TRIG;
	UldMotor3FE											: F_TRIG;
	UldMotor4RE											: R_TRIG;
	UldMotor4FE											: F_TRIG;
	UldMotor5RE											: R_TRIG;
	UldMotor5FE											: F_TRIG;

	bLoadingConveyorBusyFlag: BOOL;
	bUnloadingConveyorBusyFlag: BOOL;

	bSafetyCurtainAlarmTriggered: BOOL;
	bLdDoorSwitchCancel_TS : BOOL;
	bLdDoorSwitchForceOn_TS : BOOL;
	bUldDoorSwitchForceOn_TS : BOOL;

	tLdBasketMemoryDelayOn: TON;
	tLdBasketMemoryDelayOff: TON;

	bArm1MisshookDetectZone					: BOOL;
	bArm2MisshookDetectZone					: BOOL;

	bStn_ArmBasketNotAvailableBit							: BOOL;
	bStnBasketNotAvailableBit								: BOOL;
	bStnBasketNotAvailableBitForTempChanged				: BOOL;
	bStn6_10BasketNotAvailableBit							: BOOL;

	bLdConfirm_ConveyorNotAvailableBit	: BOOL;
	bLdTransfer_ConveyorNotAvailableBit	: BOOL;
	bAutoShutDownEnBit					: BOOL;

	bMainOnOffBuff						:BOOL;
	bAutoPreparationPbBuff				:BOOL;
	bAutoOriginPbBuff						:BOOL;
	bAutoStartPbBuff						:BOOL;

	bMainOnOff							: BOOL;
	bAutoPreparationPb      				: BOOL;
	bAutoPreparationInt	      				: BOOL;
	bAutoPreparationDone					: BOOL;
	bAutoOriginPb						: BOOL;
	bAutoOriginDone						: BOOL;
	bAutoStartPb							: BOOL;
	bAutoStartPbInt						: BOOL;
	bBasketConfirmEn						: BOOL;

(*Batch Control Mode*)
	bAutoPreparationDoneBatchMode		: BOOL;

	bAutoPreparationIntRE					: R_TRIG;

	bMainOnOffRE						: R_TRIG;
	bMainOnOffFE						: F_TRIG;
	bAutoOriginFE						: F_TRIG;
	bArmJogEnableFE					: F_TRIG;
	bAutoStartFE							: F_TRIG;
	bAutoStartRE							: R_TRIG;

	bRecipeModeOnFE					: F_TRIG;

	PowerOnDelay 							: TON;

	tSafetyCurtain1stRstTimer					: TON;
	tSafetyCurtainDelayfor2ndRstTimer			: TON;
	tSafetyCurtain2ndRstTimer					: TON;
	tSafetyCurtainReadyTimer					: TON;

	bAlarmReset_TS							: BOOL;
	bBuzzerReset_TS							: BOOL;
	bInternal_AlarmReset					: BOOL;
	bInternal_BuzzerReset					: BOOL;
	EmergencyStop							: BOOL;

	bIndusoftStart							: BOOL;
	ManualPageEnable						: BOOL;
	indusoftManual							: BOOL;
                                        	
	bAllowLoadingBasketIn					: BOOL;
	bREFE_StopLoadingBasket 				: BOOL;
                                        	
	bAutoModeLock							: BOOL;
                                        	
	bRecipeSaveInd 							: BOOL;
	bRecipeLoadInd 							: BOOL;
	bRecipeClearInd							: BOOL;     // Recipe Clear Ind For Product Recipe
	bRecipeClearInd_SSER					: BOOL;
	bRecipeClearInd_SSUR					: BOOL;
	bRecipeLoadInternal						: BOOL;
	

	iCurrentTactTime						: INT;
	iActTactTime							: INT;

(* xxxxxxxxxxxxxxxxxxxxxxxxxxxxxxx  UPS - Internal Used xxxxxxxxxxxxxxxxxxxxxxxxxxxxxxx*)
(*========================================================================*)

	bGetUpsStatusEn						: BOOL := TRUE;
	bGetUpsStatusValid					: BOOL;
	bGetUpsStatusError					: BOOL;
	udiGetUpsStatusErrID					: UDINT;
	UpsStatus							: ST_UPSStatus;

(* xxxxxxxxxxxxxxxxxxxxxxxxxxxxxxx  UPS - External Used xxxxxxxxxxxxxxxxxxxxxxxxxxxxxxx*)
(*========================================================================*)
	(* --- Alarm --- *)
	bDCPowerUnknownStatusAlarm			: BOOL;
	bBatteryUnknownStatusAlarm			: BOOL;
	bUpsCommUnknownStatusAlarm		: BOOL;
	bBatteryReplacementRequestAlarm		: BOOL;
	bUpsCommErrorAlarm					: BOOL;
	(* --- Status --- *)
	bDCPowerModeActivated				: BOOL;
	bBatteryModeActivated				: BOOL;
	bUpsCommOkFlag					: BOOL;

	timeNow: TIMESTRUCT;

END_VAR

// ---- GVLs/General_Ctrl/Global_Variables_General_Fix.TcGVL
{attribute 'Tc2GvlVarNames'}
VAR_GLOBAL

(* xxxxxxxxxxxxxxxxxxxxxxxxxxxxx Machine Time Counter xxxxxxxxxxxxxxxxxxxxxxxxxxxxx*)
(*========================================================================*)

	bMachineOnTimeRstPB_JKS							: BOOL;
	bMachineOnTimeRstPB_Customer						: BOOL;

	bMachineRunningTimeRstPB_JKS						: BOOL;
	bMachineRunningTimeRstPB_Customer					: BOOL;

(* xxxxxxxxxxxxxxxxxxxxxxxxxxxxxxxx Basket Totalizer xxxxxxxxxxxxxxxxxxxxxxxxxxxxxxxx*)
(*========================================================================*)

	bBasketTotalizerResetPB_JKS							: BOOL;
	bBasketTotalizerResetPB_Customer						: BOOL;
	bBasketTotalizerResetPB_User							: BOOL;
	bBasketTotalizerResetPB_Daily							: BOOL;

	ARbStnBasketTotalizerResetPB							: ARRAY [1..iStnQty] OF BOOL;
	ARbStnBasketCounter1stLimitAlarm						: ARRAY [1..iStnQty] OF BOOL;
	ARbStnBasketCounter2ndLimitAlarm						: ARRAY [1..iStnQty] OF BOOL;

	bBasketTotalizerResetPB_JKSPreviousLog				: BOOL;
	bBasketTotalizerResetPB_CustomerPreviousLog			: BOOL;
	bBasketTotalizerResetPB_UserPreviousLog				: BOOL;
	bBasketTotalizerResetPB_DailyPreviousLog				: BOOL;

	bBasketTotalizerResetPB_Daily1st						: BOOL;
	bBasketTotalizerResetPB_Daily2nd						: BOOL;
	bBasketTotalizerResetPB_Daily1stPreviousLog			: BOOL;
	bBasketTotalizerResetPB_Daily2ndPreviousLog			: BOOL;

(* xxxxxxxxxxxxxxxxxxxxxxxx Machine Shut Down Operation Control xxxxxxxxxxxxxxxxxxxxxxxx*)
(*========================================================================*)

	bSystemError											: BOOL;

(* xxxxxxxxxxxxxxxxxxxxxxxx BasketInfoManager xxxxxxxxxxxxxxxxxxxxxxxx*)
(*========================================================================*)

	fbBasketInfoManagerCfm_LDCV : ARRAY [0..iLdStnQty, 0..iCvLdQty] OF fbV2_BasketInfoManager;
	fbBasketInfoManagerTrf_LDCV : ARRAY [0..iLdStnQty, 0..iCvLdQty] OF fbV2_BasketInfoManager;
	fbBasketInfoManagerCfm_ULDCV : ARRAY [0..iUldStnQty, 0..iCvUldQty] OF fbV2_BasketInfoManager;
	fbBasketInfoManagerTrf_ULDCV : ARRAY [0..iUldStnQty, 0..iCvUldQty] OF fbV2_BasketInfoManager;

	fbBasketInfoManagerCfm_LD : ARRAY [0..iLdStnQty] OF fbV2_BasketInfoManager;
	fbBasketInfoManagerTrf_LD : ARRAY [0..iLdStnQty] OF fbV2_BasketInfoManager;
	fbBasketInfoManagerCfm_ULD : ARRAY [0..iUldStnQty] OF fbV2_BasketInfoManager;
	fbBasketInfoManagerTrf_ULD : ARRAY [0..iUldStnQty] OF fbV2_BasketInfoManager;

	fbBasketInfoManagerCfm_STN : ARRAY [0..iStnQty] OF fbV2_BasketInfoManager;
	fbBasketInfoManagerCfm_ARM : ARRAY [0..iArmQty] OF fbV2_BasketInfoManager;

END_VAR

// ---- GVLs/General_Ctrl/Global_Variables_General_Persistent.TcGVL
{attribute 'Tc2GvlVarNames'}
VAR_GLOBAL PERSISTENT

(* xxxxxxxxxxxxxxxxxxxxxxxxxxxxx Machine Time Counter xxxxxxxxxxxxxxxxxxxxxxxxxxxxx*)
(*========================================================================*)

	ARfbMachineTimeCounter								: ARRAY [1..4] OF fbMachineTimeCounter;

	ARfbVacPumpOnTimeCounter							: ARRAY [1..iStnQty] OF fbVacuumPumpTimeCounter;
	ARfbVacuumPump_Routine								: ARRAY [1..iStnQty] OF fbV2_EquipmentServiceCounter_Day;
	ARfbVacuumPump_Major								: ARRAY [1..iStnQty] OF fbV2_EquipmentServiceCounter_Day;

	fbPreparationTotalTimeCounter							: fbPreparationTotalTimeCounter;

	sMachineOnTime_JKS									: STRING(50);
	sMachineOnTime_Customer							: STRING(50);

	sMachineRunningTime_JKS							: STRING(50);
	sMachineRunningTime_Customer						: STRING(50);

	sMachinePreparationCurrentTime						: STRING(50);
	sMachinePreparationPreviousTime						: STRING(50);

(* xxxxxxxxxxxxxxxxxxxxxxxxxxxxxxxx Basket Totalizer xxxxxxxxxxxxxxxxxxxxxxxxxxxxxxxx*)
(*========================================================================*)

	ARfbBasketTotalizer									: ARRAY [1..6] OF fbBasketTotalizer;
	ARfbStnBasketTotalizer								: ARRAY [1..iStnQty] OF fbStnBasketTotalizer;

	diTotalBasketQty_JKS									: DINT;
	diTotalBasketQty_Customer							: DINT;
	diTotalBasketQty_User								: DINT;
	diTotalBasketQty_Daily								: DINT;
	diTotalBasketQty_Daily1st								: DINT;
	diTotalBasketQty_Daily2nd								: DINT;

	diPreviousTotalBasketQtyLog_Daily						: DINT;
	diPreviousTotalBasketQtyLog_Daily1st					: DINT;
	diPreviousTotalBasketQtyLog_Daily2nd					: DINT;

	ARdiTotalStnBasketQty								: ARRAY [1..iStnQty] OF DINT;
	ARdiStnBasketCounter1stLimitSV						: ARRAY [1..iStnQty] OF DINT;
	ARdiStnBasketCounter2ndLimitSV						: ARRAY [1..iStnQty] OF DINT;

	wZeroValue											: WORD := 0;
	wAutoStartHourSV_Daily								: WORD;
	wAutoStartHourSV_Daily1st								: WORD;
	wAutoStartHourSV_Daily2nd							: WORD;

	wAutoDurationHourSV_JKS								: WORD;
	wAutoDurationHourSV_Customer						: WORD;
	wAutoDurationHourSV_User							: WORD;
	wAutoDurationHourSV_Daily							: WORD;
	wAutoDurationHourSV_Daily1st							: WORD;
	wAutoDurationHourSV_Daily2nd							: WORD;

(* xxxxxxxxxxxxxxxxxxxxxx Machine Shut Down Operation Control xxxxxxxxxxxxxxxxxxxxxx*)
(*========================================================================*)

	wShutDownYear										: WORD;
	wShutDownMonth										: WORD;
	wShutDownDay										: WORD;

	bMcShutDownDisable									: BOOL;

(* xxxxxxxxxxxxxxxxxxxxxxxxxxxxx Vacuum Pump Time Counter xxxxxxxxxxxxxxxxxxxxxxxxxxxxx*)
(*========================================================================*)

	ARsVacuumPumpRunningTime							: ARRAY [1..iStnQty] OF STRING(50);

(* xxxxxxxxxxxxxxxxxxxxxxxxxxxxxxx User Password Used xxxxxxxxxxxxxxxxxxxxxxxxxxxxxxx*)
(*========================================================================*)

	UserPassword										: ARRAY [0..7] OF STRING;
	UserName											: ARRAY [0..7] OF wSTRING;
	UserLogin											: ARRAY [0..7] OF BOOL;

(*XML Prev Recipe No*)
	iPrevrecipeNo	:INT;
	iAutoPrevRecipeMode:INT;

END_VAR

// ---- GVLs/GVL3/GVL_Analog.TcGVL
{attribute 'Tc2GvlVarNames'}
VAR_GLOBAL CONSTANT
	
iTempCtrlQty 			: INT := 9; // Quantity of Temperature Control
iPressureCtrlQty		: INT := 8; // Quantity of Pressure Control
//iPHQty				: INT := 1; // Quantity of PH
//iFlowQty				: INT := 7; // Quantity of Flow Control
iConductivity			: INT := 8; // Quantity of Conductivity Control
//iVacuum				: INT := 1; // Quantity of Vacuum Control

END_VAR

VAR_GLOBAL
	
(* xxxxxxxxxxxxxxxxxxxxxxxxxxxxxxxx Analog Mapping xxxxxxxxxxxxxxxxxxxxxxxxxxxxxxxx*)
(*========================================================================*)

	ANI1_1	AT %I*	: INT; // STN 01 ULTRASONIC GENERATOR (LEFT &RIGHT) POWER SIGNAL
	ANI1_2	AT %I*	: INT; // STN 01 ULTRASONIC GENERATOR (BOTTOM) POWER SIGNAL
	ANI1_3	AT %I*	: INT; // STN 02 ULTRASONIC GENERATOR (LEFT &RIGHT) POWER SIGNAL
	ANI1_4	AT %I*	: INT; // STN 02 ULTRASONIC GENERATOR (BOTTOM) POWER SIGNAL
  
	ANI2_1	AT %I*	: INT; // STN 03 ULTRASONIC GENERATOR (LEFT &RIGHT) POWER SIGNAL
	ANI2_2	AT %I*	: INT; // STN 03 ULTRASONIC GENERATOR (BOTTOM) POWER SIGNAL
	ANI2_3	AT %I*	: INT; // STN 04 ULTRASONIC GENERATOR (LEFT &RIGHT) POWER SIGNAL
	ANI2_4	AT %I*	: INT; // STN 04 ULTRASONIC GENERATOR (BOTTOM) POWER SIGNAL

	ANI3_1	AT %I*	: INT; // STN 05 ULTRASONIC GENERATOR (BOTTOM) POWER SIGNAL
	ANI3_2	AT %I*	: INT; // STN 06 PROCESS TANK VACUUM SIGNAL
	ANI3_3	AT %I*	: INT; // RESERVED
	ANI3_4	AT %I*	: INT; // RESERVED
	
	ANI4_1	AT %I*	: INT; // STN 01 PROCESS TANK PRESSURE SWITCH SIGNAL
	ANI4_2	AT %I*	: INT; // STN 02 PROCESS TANK PRESSURE SWITCH SIGNAL
	ANI4_3	AT %I*	: INT; // RESERVED  
	ANI4_4	AT %I*	: INT; // RESERVED  
	
	ANI5_1	AT %I*	: INT; // STN 03 PROCESS TANK PRESSURE SWITCH SIGNAL
	ANI5_2	AT %I*	: INT; // STN 04 PROCESS TANK PRESSURE SWITCH SIGNAL
	ANI5_3	AT %I*	: INT; // RESERVED
	ANI5_4	AT %I*	: INT; // RESERVED
	
	ANI6_1	AT %I*	: INT; // STN 05 PROCESS TANK PRESSURE SWITCH SIGNAL
	ANI6_2	AT %I*	: INT; // STN 05 PROCESS TANK CONDUCTIVITY SIGNAL 
	ANI6_3	AT %I*	: INT; // RESERVED 
	ANI6_4	AT %I*	: INT; // RESERVED 
	
	RTD1_1  AT %I* 	: INT; // STN 01 PROCESS TANK PT100 RTD
	RTD1_2  AT %I* 	: INT; // STN 02 PROCESS TANK PT100 RTD
	RTD1_3  AT %I* 	: INT; // RESERVED                     
	RTD1_4  AT %I* 	: INT; // RESERVED                     
	
	RTD2_1  AT %I* 	: INT; // STN 03 PROCESS TANK PT100 RTD
	RTD2_2  AT %I* 	: INT; // STN 04 PROCESS TANK PT100 RTD
	RTD2_3  AT %I* 	: INT; // RESERVED
	RTD2_4  AT %I* 	: INT; // RESERVED
	
	RTD3_1  AT %I*	: INT; // STN 05 PROCESS TANK PT100 RTD
	RTD3_2  AT %I*	: INT; // RESERVED                   
	
	TYK1_1	AT %I*	: INT; // STN 06 PROCESS TANK TYPE-K THERMOCOUPLE
	TYK1_2	AT %I*	: INT; // RESERVED                               
	
//	TYK2_1	AT %I*	: INT; // STN 09 LEFT TOP HEATER TYPE-K THERMOCOUPLE    
//	TYK2_2	AT %I*	: INT; // STN 09 LEFT BOTTOM HEATER TYPE-K THERMOCOUPLE 
//	TYK2_3	AT %I*	: INT; // STN 09 RIGHT TOP HEATER TYPE-K THERMOCOUPLE   
//	TYK2_4	AT %I*	: INT; // STN 09 RIGHT BOTTOM HEATER TYPE-K THERMOCOUPLE
	
//	COM1_1	AT %I*	: INT; // STN 01 ULTRASONIC GENERATOR MODBUS SIGNAL
//	COM1_2	AT %I*	: INT; // STN 02 ULTRASONIC GENERATOR MODBUS SIGNAL
//	COM1_3	AT %I*	: INT; // STN 03 ULTRASONIC GENERATOR MODBUS SIGNAL
//	COM1_4	AT %I*	: INT; // STN 04 ULTRASONIC GENERATOR MODBUS SIGNAL
//	COM1_5	AT %I*	: INT; // STN 05 ULTRASONIC GENERATOR MODBUS SIGNAL
//	COM1_6	AT %I*	: INT; // STN 06 ULTRASONIC GENERATOR MODBUS SIGNAL
	
//	COM2_1	AT %I*	: INT; // STN 03 MEGASONIC GENERATOR 01 MODBUS SIGNAL (-16U1)
//	COM2_2	AT %I*	: INT; // STN 03 MEGASONIC GENERATOR 02 MODBUS SIGNAL (-17U1)
//	COM2_3	AT %I*	: INT; // STN 06 MEGASONIC GENERATOR 01 MODBUS SIGNAL (-18U1)
//	COM2_4	AT %I*	: INT; // STN 06 MEGASONIC GENERATOR 02 MODBUS SIGNAL (-19U1)
//	COM2_5	AT %I*	: INT; // STN 06 MEGASONIC GENERATOR 03 MODBUS SIGNAL (-20U1)
	
	(*ANALOG OUTPUT*)

	ANO1_1   		AT %Q* : INT; // STN 01 ULTRASONIC GENERATOR (LEFT & RIGHT) POWER SIGNAL
	ANO1_2   		AT %Q* : INT; // STN 01 ULTRASONIC GENERATOR (BOTTOM) POWER SIGNAL
	ANO1_3   		AT %Q* : INT; // STN 02 ULTRASONIC GENERATOR (LEFT & RIGHT) POWER SIGNAL
	ANO1_4   		AT %Q* : INT; // STN 02 ULTRASONIC GENERATOR (BOTTOM) POWER SIGNAL
	
	ANO2_1   		AT %Q* : INT; // STN 03 ULTRASONIC GENERATOR (LEFT & RIGHT) POWER SIGNAL
	ANO2_2   		AT %Q* : INT; // STN 03 ULTRASONIC GENERATOR (BOTTOM) POWER SIGNAL
	ANO2_3   		AT %Q* : INT; // STN 04 ULTRASONIC GENERATOR (LEFT & RIGHT) POWER SIGNAL
	ANO2_4   		AT %Q* : INT; // STN 04 ULTRASONIC GENERATOR (BOTTOM) POWER SIGNAL
                                 
    ANO3_1   		AT %Q* : INT; // STN 05 ULTRASONIC GENERATOR (BOTTOM) POWER SIGNAL
	ANO3_2   		AT %Q* : INT; // RESERVED                                           
	
//	BAC1_1	AT %I*	: INT; // LOADING BARCODE READER

//(* ENCODER MAPPING*)

//	bIN_VertSetCounterDone 		AT %I* 	: ARRAY [1..iArmQty] OF BOOL;
//	udIN_VertCounterValue 		AT %I* 	: ARRAY [1..iArmQty] OF UDINT;

//	bOUT_VertSetCounterEn 		AT %Q* 	: ARRAY [1..iArmQty] OF BOOL;
//	udOUT_VertSetCounterValue 	AT %Q* 	: ARRAY [1..iArmQty] OF UDINT;

//	bIN_HorzSetCounterDone 		AT %I* 	: ARRAY [1..iArmQty] OF BOOL;
//	udIN_HorzCounterValue 		AT %I* 	: ARRAY [1..iArmQty] OF UDINT;

//	bOUT_HorzSetCounterEn 		AT %Q* 	: ARRAY [1..iArmQty] OF BOOL;
//	udOUT_HorzSetCounterValue 	AT %Q* 	: ARRAY [1..iArmQty] OF UDINT;

(* xxxxxxxxxxxxxxxxxxxxxxxxxxxxxxxx Temperature Ctrl xxxxxxxxxxxxxxxxxxxxxxxxxxxxxxxx*)
(*========================================================================*)

//	ARfb3TempControl								: ARRAY [0..iTempCtrlQty] OF FB3_TempControl;
//	ARrTempPresentValue_PV							: ARRAY [0..iTempCtrlQty] OF REAL;
//	ARbTempOnOff									: ARRAY [0..iTempCtrlQty] OF BOOL;
//	ARbTempReady									: ARRAY [0..iTempCtrlQty] OF BOOL;
//	ARbTempHighAlarm								: ARRAY [0..iTempCtrlQty] OF BOOL;
//	ARbTemp1stLimitAlarm							: ARRAY [0..iTempCtrlQty] OF BOOL;
//	ARbTempPreparationNoRdyAlarm					: ARRAY [0..iTempCtrlQty] OF BOOL;
//	ARrDefaultStationTemperatureSV					: ARRAY [0..C_iProcessStnQty] OF REAL;
//	ARbTempWarningLowAlarm							: ARRAY [0..iTempCtrlQty] OF BOOL;
//	ARbTempWarningHighAlarm							: ARRAY [0..iTempCtrlQty] OF BOOL;
//	ARbTempAlarmLowAlarm							: ARRAY [0..iTempCtrlQty] OF BOOL;
//	ARbTempAlarmHighAlarm							: ARRAY [0..iTempCtrlQty] OF BOOL;
	
(* xxxxxxxxxxxxxxxxxxxxxxxxxxxxxxxx Pressure Ctrl xxxxxxxxxxxxxxxxxxxxxxxxxxxxxxxx*)
(*========================================================================*)

//	ARfb3PressureControl							: ARRAY [0..iPressureCtrlQty] OF FB3_RawRatioConversionReal;
//	ARrPressurePresentValue_PV						: ARRAY [0..iPressureCtrlQty] OF REAL;
//	ARbPressureLowAlarm								: ARRAY [0..iPressureCtrlQty] OF BOOL;
//	ARbPressureHighAlarm							: ARRAY [0..iPressureCtrlQty] OF BOOL;	
//	ARbPressureWarningLowAlarm						: ARRAY [0..iPressureCtrlQty] OF BOOL;
//	ARbPressureWarningHighAlarm						: ARRAY [0..iPressureCtrlQty] OF BOOL;
//	ARbPressureAlarmLowAlarm						: ARRAY [0..iPressureCtrlQty] OF BOOL;
//	ARbPressureAlarmHighAlarm						: ARRAY [0..iPressureCtrlQty] OF BOOL;
	
//	bStn5HeaterOff									: BOOL;

	
(* xxxxxxxxxxxxxxxxxxxxxxxxxxxxxxxx PH Ctrl xxxxxxxxxxxxxxxxxxxxxxxxxxxxxxxx*)
(*========================================================================*)

//	ARfb3PHControl									: ARRAY [0..iPHQty] OF FB3_RawRatioConversionReal;
//	ARrPHPresentValue_PV							: ARRAY [0..iPHQty] OF REAL;
//	ARbPHLowAlarm									: ARRAY [0..iPHQty] OF BOOL;
//	ARbPHHighAlarm									: ARRAY [0..iPHQty] OF BOOL;	
//	ARbPHWarningLowAlarm							: ARRAY [0..iPHQty] OF BOOL;
//	ARbPHWarningHighAlarm							: ARRAY [0..iPHQty] OF BOOL;
//	ARbPHAlarmLowAlarm								: ARRAY [0..iPHQty] OF BOOL;
//	ARbPHAlarmHighAlarm								: ARRAY [0..iPHQty] OF BOOL;
	
(* xxxxxxxxxxxxxxxxxxxxxxxxxxxxxxxx Flow Ctrl xxxxxxxxxxxxxxxxxxxxxxxxxxxxxxxx*)
(*========================================================================*)

//	ARfb3FlowControl								: ARRAY [0..iFlowQty] OF FB3_RawRatioConversionReal;
//	ARfb3FlowControl1								: ARRAY [0..iFlowQty] OF FB2_KeyenceVacSensorTuningkPa;
	
//	ARbFlowLowSave									: ARRAY [0..iFlowQty] OF BOOL;
//	ARbFlowHighSave									: ARRAY [0..iFlowQty] OF BOOL;
//	ARrFlowPresentValue_PV							: ARRAY [0..iFlowQty] OF REAL;
//	ARbFlowLowAlarm									: ARRAY [0..iFlowQty] OF BOOL;
//	ARbFlowHighAlarm								: ARRAY [0..iFlowQty] OF BOOL;	
//	ARbFlowWarningLowAlarm							: ARRAY [0..iFlowQty] OF BOOL;
//	ARbFlowWarningHighAlarm							: ARRAY [0..iFlowQty] OF BOOL;
//	ARbFlowAlarmLowAlarm							: ARRAY [0..iFlowQty] OF BOOL;
//	ARbFlowAlarmHighAlarm							: ARRAY [0..iFlowQty] OF BOOL;
	
(* xxxxxxxxxxxxxxxxxxxxxxxxxxxxxxxx Conductivity Ctrl xxxxxxxxxxxxxxxxxxxxxxxxxxxxxxxx*)
(*========================================================================*)

//	ARfb3ConductivityControl						: ARRAY [0..iConductivity] OF FB3_RawRatioConversionReal;
//	ARrConductivityPresentValue_PV					: ARRAY [0..iConductivity] OF REAL;
//	ARbConductivityLowAlarm							: ARRAY [0..iConductivity] OF BOOL;
//	ARbConductivityHighAlarm						: ARRAY [0..iConductivity] OF BOOL;	
//	ARbConductivityWarningLowAlarm					: ARRAY [0..iConductivity] OF BOOL;
//	ARbConductivityWarningHighAlarm					: ARRAY [0..iConductivity] OF BOOL;
//	ARbConductivityAlarmLowAlarm					: ARRAY [0..iConductivity] OF BOOL;
//	ARbConductivityAlarmHighAlarm					: ARRAY [0..iConductivity] OF BOOL;
	
	
(* xxxxxxxxxxxxxxxxxxxxxxxxxxxxxxxx Vacuum Ctrl xxxxxxxxxxxxxxxxxxxxxxxxxxxxxxxx*)
(*========================================================================*)

//	ARfbVacuumPump_Routine							: ARRAY [0..iStnQty] OF fbV2_EquipmentServiceCounter_Day;
//	ARfbVacuumPump_Major							: ARRAY [0..iStnQty] OF fbV2_EquipmentServiceCounter_Day;
//	fbVacuumCalibration								: ARRAY [0..iVacuum] OF FB2_KeyenceVacSensorTuningkPa;
//	ARrVacuumPresentValue_PV						: ARRAY [0..iVacuum] OF REAL;
//	ARbVacuumLowSignal								: ARRAY [0..iVacuum] OF BOOL;
//	ARbVacuumHighSignal								: ARRAY [0..iVacuum] OF BOOL;
//	ARbVacuumLowSave								: ARRAY [0..iVacuum] OF BOOL;
//	ARbVacuumHighSave								: ARRAY [0..iVacuum] OF BOOL;	
	
END_VAR

// ---- GVLs/GVL3/GVL_Deactivate_Persistent.TcGVL
{attribute 'Tc2GvlVarNames'}
VAR_GLOBAL PERSISTENT
	
	DE10000  : BOOL;   // EMERGENCY STOP SAFETY RELAY - RESET  (-250K3)              
	DE10001  : BOOL;   // STN 01 ULTRASONIC GENERATOR FREQUENCY CHANGE (-10U1)       
	DE10002  : BOOL;   // STN 02 ULTRASONIC GENERATOR FREQUENCY CHANGE (-11U1)       
	DE10003  : BOOL;   // STN 04 ULTRASONIC GENERATOR FREQUENCY CHANGE (-12U1)       
	DE10004  : BOOL;   // STN 05 ULTRASONIC GENERATOR FREQUENCY CHANGE (-13U1)       
	DE10005  : BOOL;   // STN 07 ULTRASONIC GENERATOR FREQUENCY CHANGE (-14U1)       
	DE10006  : BOOL;   // STN 08 ULTRASONIC GENERATOR FREQUENCY CHANGE (-15U1)       
	DE10007  : BOOL;   // STN 09 SLOW PULL MECHANISM SERVO MOTOR - ERROR STOP (-42U1)
	DE10008  : BOOL;   // ARM 01 HORIZONTAL SERVO MOTOR - ERROR STOP (-40U1)         
	DE10009  : BOOL;   // ARM 01 VERTICAL SERVO MOTOR - ERROR STOP (-41U1)           
	DE10010  : BOOL;   // RESERVED                                                   
	DE10011  : BOOL;   // RESERVED                                                   
	DE10012  : BOOL;   // RESERVED                                                   
	DE10013  : BOOL;   // RESERVED                                                   
	DE10014  : BOOL;   // RESERVED                                                   
	DE10015  : BOOL;   // RESERVED                                                   
	
	DE10100  : BOOL;   // STN 01 ULTRASONIC GENERATOR ON/OFF (-10U1)     
	DE10101  : BOOL;   // STN 02 ULTRASONIC GENERATOR ON/OFF (-11U1)     
	DE10102  : BOOL;   // STN 04 ULTRASONIC GENERATOR ON/OFF (-12U1)     
	DE10103  : BOOL;   // STN 05 ULTRASONIC GENERATOR ON/OFF (-13U1)     
	DE10104  : BOOL;   // STN 07 ULTRASONIC GENERATOR ON/OFF (-14U1)     
	DE10105  : BOOL;   // STN 08 ULTRASONIC GENERATOR ON/OFF (-15U1)     
	DE10106  : BOOL;   // STN 07 DI WATER RETURN TANK PUMP ON/OFF (-81K1)
	DE10107  : BOOL;   // STN 01 PROCESS TANK PUMP ON/OFF (-73K1)        
	DE10108  : BOOL;   // STN 02 PROCESS TANK PUMP ON/OFF (-74K1)        
	DE10109  : BOOL;   // STN 03 PROCESS TANK PUMP ON/OFF (-75K1)        
	DE10110  : BOOL;   // STN 04 PROCESS TANK PUMP ON/OFF (-76K1)        
	DE10111  : BOOL;   // STN 05 PROCESS TANK PUMP ON/OFF (-77K1)        
	DE10112  : BOOL;   // STN 06 PROCESS TANK PUMP ON/OFF (-78K1)        
	DE10113  : BOOL;   // STN 07 PROCESS TANK PUMP ON/OFF (-79K1)        
	DE10114  : BOOL;   // STN 08 PROCESS TANK PUMP ON/OFF (-80K1)        
	DE10115  : BOOL;   // STN 01 PROCESS TANK HEATER ON/OFF (-130K1)     
	
	DE10200  : BOOL;   // STN 02 PROCESS TANK HEATER ON/OFF (-131K1) 
	DE10201  : BOOL;   // STN 03 PROCESS TANK HEATER ON/OFF (-132K1) 
	DE10202  : BOOL;   // STN 04 PROCESS TANK HEATER ON/OFF (-133K1) 
	DE10203  : BOOL;   // STN 05 PROCESS TANK HEATER ON/OFF (-134K1) 
	DE10204  : BOOL;   // STN 06 PROCESS TANK HEATER ON/OFF (-135K1) 
	DE10205  : BOOL;   // STN 07 PROCESS TANK HEATER ON/OFF (-136K1) 
	DE10206  : BOOL;   // STN 08 PROCESS TANK HEATER ON/OFF (-137K1) 
	DE10207  : BOOL;   // STN 10 PROCESS TANK HEATER ON/OFF (-138K1) 
	DE10208  : BOOL;   // STN 09 - STN 10 FFU UNIT ON/OFF (-163K1)   
	DE10209  : BOOL;   // UNLOADING FFU UNIT ON/OFF (-164K1)         
	DE10210  : BOOL;   // UNLOADING CONVEYOR FFU UNIT ON/OFF (-165K1)
	DE10211  : BOOL;   // STN 09 PROCESS TANK PUMP ON/OFF (-82K1)    
	DE10212  : BOOL;   // RESERVED                                   
	DE10213  : BOOL;   // RESERVED                                   
	DE10214  : BOOL;   // RESERVED                                   
	DE10215  : BOOL;   // RESERVED                                   
	
	DE10300  : BOOL;   // STN 01 - 08 AGITATION MOTOR ON/OFF (-160K1)
	DE10301  : BOOL;   // LOADING CONVEYOR 01 ON/OFF (-170K1)        
	DE10302  : BOOL;   // LOADING CONVEYOR 02 ON/OFF (-171K1)        
	DE10303  : BOOL;   // LOADING CONVEYOR 03 ON/OFF (-172K1)        
	DE10304  : BOOL;   // LOADING CONVEYOR 04 ON/OFF (-173K1)        
	DE10305  : BOOL;   // UNLOADING CONVEYOR 01 ON/OFF (-174K1)      
	DE10306  : BOOL;   // UNLOADING CONVEYOR 02 ON/OFF (-175K1)      
	DE10307  : BOOL;   // UNLOADING CONVEYOR 03 ON/OFF (-176K1)      
	DE10308  : BOOL;   // UNLOADING CONVEYOR 04 ON/OFF (-177K1)      
	DE10309  : BOOL;   // RESERVED                                   
	DE10310  : BOOL;   // RESERVED                                   
	DE10311  : BOOL;   // RESERVED                                   
	DE10312  : BOOL;   // RESERVED                                   
	DE10313  : BOOL;   // RESERVED                                   
	DE10314  : BOOL;   // RESERVED                                   
	DE10315  : BOOL;   // RESERVED                                   
	
	DE10400  : BOOL;	
	DE10401  : BOOL;	
	DE10402  : BOOL;	
	DE10403  : BOOL;	
	DE10404  : BOOL;	
	DE10405  : BOOL;	
	DE10406  : BOOL;	
	DE10407  : BOOL;	
	DE10408  : BOOL;	
	DE10409  : BOOL;	
	DE10410  : BOOL;	
	DE10411  : BOOL;	
	DE10412  : BOOL;	
	DE10413  : BOOL;	
	DE10414  : BOOL;	
	DE10415  : BOOL;	
		
	DE11000  : BOOL;   // GENERAL ALARM RESET IND (-310S1)         
	DE11001  : BOOL;   // GENERAL BUZZER  RESET IND (-310S2)       
	DE11002  : BOOL;   // GENERAL BUZZER TONE 01 (-410H1)          
	DE11003  : BOOL;   // GENERAL BUZZER TONE 02 (-410H1)          
	DE11004  : BOOL;   // GENERAL TOWER LIGHT IND - RED (-410H2)   
	DE11005  : BOOL;   // GENERAL TOWER LIGHT IND - YELLOW (-410H2)
	DE11006  : BOOL;   // GENERAL TOWER LIGHT IND - GREEN (-410H2) 
	DE11007  : BOOL;   // IPC DC ON HOLDING RELAY (-410K1)         
	DE11008  : BOOL;   // RESERVED                                 
	DE11009  : BOOL;   // RESERVED                                 
	DE11010  : BOOL;   // RESERVED                                 
	DE11011  : BOOL;   // RESERVED                                 
	DE11012  : BOOL;   // RESERVED                                 
	DE11013  : BOOL;   // RESERVED                                 
	DE11014  : BOOL;   // RESERVED                                 
	DE11015  : BOOL;   // RESERVED                                 
	
	DE11100  : BOOL;   // STN 03 MEGASONIC GENERATOR 01 ON/OFF (-16U1)
	DE11101  : BOOL;   // STN 03 MEGASONIC GENERATOR 02 ON/OFF (-17U1)
	DE11102  : BOOL;   // STN 01 DOSING PUMP ON/OFF (-70K1)           
	DE11103  : BOOL;   // STN 03 DOSING PUMP ON/OFF (-71K1)           
	DE11104  : BOOL;   // RESERVED                                    
	DE11105  : BOOL;   // RESERVED                                    
	DE11106  : BOOL;   // RESERVED                                    
	DE11107  : BOOL;   // RESERVED                                    
	DE11108  : BOOL;   // RESERVED                                    
	DE11109  : BOOL;   // RESERVED                                    
	DE11110  : BOOL;   // RESERVED                                    
	DE11111  : BOOL;   // RESERVED                                    
	DE11112  : BOOL;   // RESERVED                                    
	DE11113  : BOOL;   // RESERVED                                    
	DE11114  : BOOL;   // RESERVED                                    
	DE11115  : BOOL;   // RESERVED                                    
	
	DE12000  : BOOL;   // STN 05 DOSING PUMP ON/OFF (-72K1)           
	DE12001  : BOOL;   // STN 06 MEGASONIC GENERATOR 01 ON/OFF (-18U1)
	DE12002  : BOOL;   // STN 06 MEGASONIC GENERATOR 02 ON/OFF (-19U1)
	DE12003  : BOOL;   // STN 06 MEGASONIC GENERATOR 03 ON/OFF (-20U1)
	DE12004  : BOOL;   // RESERVED                                    
	DE12005  : BOOL;   // RESERVED                                    
	DE12006  : BOOL;   // RESERVED                                    
	DE12007  : BOOL;   // RESERVED                                    
	DE12008  : BOOL;   // RESERVED                                    
	DE12009  : BOOL;   // RESERVED                                    
	DE12010  : BOOL;   // RESERVED                                    
	DE12011  : BOOL;   // RESERVED                                    
	DE12012  : BOOL;   // RESERVED                                    
	DE12013  : BOOL;   // RESERVED                                    
	DE12014  : BOOL;   // RESERVED                                    
	DE12015  : BOOL;   // RESERVED                                    
	
	DE13000  : BOOL;   // STN 01 DIW INCOMING SUPPLY AV1-1 (-430Y1)  
	DE13001  : BOOL;   // STN 01 OVERFLOW SUCTION AV1-2 (-430Y2)     
	DE13002  : BOOL;   // STN 02 ROW INCOMING SUPPLY AV2-1 (-430Y3)  
	DE13003  : BOOL;   // STN 03 DIW INCOMING SUPPLY AV3-1 (-430Y4)  
	DE13004  : BOOL;   // STN 03 OVERFLOW SUCTION AV3-2 (-430Y5)     
	DE13005  : BOOL;   // STN 03 CHILLED WATER SUPPLY AV3-3 (-430Y6) 
	DE13006  : BOOL;   // STN 04 ROW INCOMING SUPPLY AV4-1 (-430Y7)  
	DE13007  : BOOL;   // STN 05 DIW INCOMING SUPPLY AV5-1 (-430Y8)  
	DE13008  : BOOL;   // STN 05 OVERFLOW SUCTION AV5-2 (-430Y9)     
	DE13009  : BOOL;   // STN 06 ROW INCOMING SUPPLY AV6-1 (-430Y10) 
	DE13010  : BOOL;   // STN 06 CHILLED WATER SUPPLY AV6-2 (-430Y11)
	DE13011  : BOOL;   // STN 07 DIW INCOMING SUPPLY AV7-1 (-430Y12) 
	DE13012  : BOOL;   // STN 08 DIW INCOMING SUPPLY AV8-1 (-430Y13) 
	DE13013  : BOOL;   // STN 09 DIW INCOMING SUPPLY AV9-1 (-430Y14) 
	DE13014  : BOOL;   // DIW MAIN INCOMING SUPPLY AVINC-1 (-430Y15) 
	DE13015  : BOOL;   // ROW MAIN INCOMING SUPPLY AVINC-2 (-430Y16) 
	
	DE13100  : BOOL;   // UNLOADING SHUTTER DOOR - OPEN (-431Y1)          
	DE13101  : BOOL;   // UNLOADING SHUTTER DOOR - CLOSE (-431Y2)         
	DE13102  : BOOL;   // UNLOADING CONVEYOR SHUTTER DOOR - OPEN (-431Y3) 
	DE13103  : BOOL;   // UNLOADING CONVEYOR SHUTTER DOOR - CLOSE (-431Y4)
	DE13104  : BOOL;   // RESERVED                                        
	DE13105  : BOOL;   // RESERVED                                        
	DE13106  : BOOL;   // RESERVED                                        
	DE13107  : BOOL;   // RESERVED                                        
	DE13108  : BOOL;   // RESERVED                                        
	DE13109  : BOOL;   // RESERVED                                        
	DE13110  : BOOL;   // RESERVED                                        
	DE13111  : BOOL;   // RESERVED                                        
	DE13112  : BOOL;   // RESERVED                                        
	DE13113  : BOOL;   // RESERVED                                        
	DE13114  : BOOL;   // RESERVED                                        
	DE13115  : BOOL;   // RESERVED                                        

//	bDeactivateMagneticSwitchDoorAlarm	: BOOL;
//	bDeactivateSlidingWindowAlarm		: BOOL;	
//	ARbDeactivateMissHookAlarm			: ARRAY [0..C_iMcArmHookQty] OF BOOL;
//	ARbDeactivateArmCrashAlarm			: ARRAY [0..C_iMcArmHookQty] OF BOOL;
	
	
END_VAR

// ---- GVLs/GVL3/GVL_Event_Module.TcGVL
VAR_GLOBAL
	fb3EventModule							:FB3_EventModule;
	bEventRstPBPhysicalInput				: BOOL;
	bBuzzerRstPBPhysicalInput				: BOOL;
	bAcknowdgePBPhysicalInput				: BOOL;
	//bEventRstPB							: BOOL;
	//bBuzerRstPB							: BOOL;
	//bAcknowledgePB						: BOOL;
	bAcknowledgeEnable						: BOOL; 
	tPowerUpDelayTime						: TIME;
	//eHmiLanguage							: E_HmiLanguage; 
	bActiveEventDisplay_ScrollUp			: BOOL;
	bActiveEventDisplay_ScrollDown			: BOOL;
	bHistoryEventDisplay_ScrollUp			: BOOL;
	bHistoryEventDisplay_ScrollDown			: BOOL;	
	bCautionEventOccuredFlag 				: BOOL;
	bWarningEventOccuredFlag 				: BOOL;
	bErrorEventOccuredFlag 					: BOOL;
	bEventOccuredFlag						: BOOL;
	iActiveCautionEventCount				: INT;
	iActiveWarningEventCount 				: INT;
	iActiveErrorEventCount	 				: INT;
	bBuzzerOutput							: BOOL;	
END_VAR

// ---- GVLs/GVL3/LIB_GVL_EVENT.TcGVL
{attribute 'Tc2GvlVarNames'}

VAR_GLOBAL

	ARdsEventActiveLog						: ARRAY [0..C_iEventActiveLogQty] 						OF DS_Event;	// Keep certain quantity of Active Event Log to allow view in HMI
	ARdsEventActiveDisplay					: ARRAY [1..C_iEventActiveDisplayQty] 					OF DS_ActiveEventDisplay; // compiled Event info with Active Language Reference	
	ARdsEventHistoryDisplay					: ARRAY [1..C_iEventHistoryDisplayQty] 					OF DS_HistoryEventDisplay; // compiled Event info with Active Language Reference	

	ARdsEventCtrl		 					: ARRAY [0..C_iEventQty] 								OF DS_EventControl ; 				//XML_AutoRO_ManualRW	// Signal, Timer and Output variable for Event	

//	ARdsEventActiveLog_Empty				: ARRAY [0..C_iEventActiveLogQty] 						OF DS_Event;	// Keep certain quantity of Active Event Log to allow view in HMI

	dsEventCtrlEmpty						: DS_EventControl;
	dsEventActiveDisplayEmpty				: DS_ActiveEventDisplay;
	dsEventHistoryDisplayEmpty				: DS_HistoryEventDisplay;
	dsEventActiveLogEmpty					: DS_Event;																

	dsEventHistoryLogEmpty					: DS_EventHistory;
	dsEventHistoryLogToFileEmpty			: DS_EventHistory;




END_VAR

VAR_GLOBAL PERSISTENT
	


	AR2dsEventDescriptionCausedRemedy		: ARRAY [1..C_iLanguageQty] OF ARRAY [0..C_iEventQty] 	OF DS_EventDescriptionCausedRemedy; //XML_AutoRO_ManualRW, keep multi-language info

	
	ARdsEventHistoryLog		 				: ARRAY [0..C_iEventHistoryLogQty] 						OF DS_EventHistory; // Keep certain quantity of History Event Log to allow view in HMI
//	ARdsEventHistoryLog_Empty 				: ARRAY [0..C_iEventHistoryLogQty] 						OF DS_EventHistory; // Keep certain quantity of History Event Log to allow view in HMI

//	ARdsEventHistoryLogToFile 				: ARRAY [0..C_iRingBufferQty] 							OF DS_EventHistory;  // Buffer data to get ready to store in XML/CSV	
END_VAR

// ---- GVLs/GVL3/LIB_GVL_GENERAL.TcGVL
{attribute 'Tc2GvlVarNames'}
VAR_GLOBAL




// Clock Timer Counter
	dsLocalSystemTimeML 						: DS_LocalSystemTime;	// Multi-Language Support
	SysTime										: TIMESTRUCT;			// System Time (Structure)
	sSysTime									: STRING(50);

	bClockPulse_1Sec							: BOOL; // its a Pulse, so no need to add R_TRIG
	bClockPulse_0_5Sec							: BOOL; // its a Pulse, so no need to add R_TRIG
	bClockPulse_0_1Sec							: BOOL; // its a Pulse, so no need to add R_TRIG
	bClockPulse_10ms							: BOOL; // its a Pulse, so no need to add R_TRIG
	bClockBlink_1Sec							: BOOL; // 0.5Sec ON <-> 0.5Sec OFF
	
// HMI Related	
//	bSavePB_Recipe								: BOOL;
//	bSaveAndUpdateAllCheckBox					: BOOL;
//	bLoadPB_Recipe								: BOOL; (* For PLC Used only *)
//	bReloadPB_Recipe							: BOOL; 

//	bSavePB_RecipeRE							: R_TRIG;
//	bLoadPB_RecipeRE							: R_TRIG;	
//	bReloadPB_RecipeRE							: R_TRIG;	
	
//	bSavePB_RecipeFE							: F_TRIG;	
//	bLoadPB_RecipeFE							: F_TRIG;		
//	bReloadPB_RecipeFE							: F_TRIG;		
		
	
//	bSavePBInd_Recipe							: BOOL;
//	bLoadPBInd_Recipe							: BOOL;
//	bReloadPBInd_Recipe							: BOOL;	

//	bHmiInitialisationFlag						: BOOL;
//	bHmiInitialisationPulse						: BOOL;

//	bHmi_ActiveUsernameChangedPulse				: BOOL;	


//	XML Manually Import and Export - FB3_XmlSvrRW_Recipe
(**)	bManualRecipe_ImportSt						: BOOL;
(**)	bManualRecipe_ImportBusyFlag				: BOOL;
(**)	bManualRecipe_ImportDoneFlag				: BOOL;
(**)	bManualRecipe_ImportErrFlag					: BOOL;
		udManualRecipe_ImportErrId					: UDINT;

(**)	bManualRecipe_ExportSt						: BOOL;
(**)	bManualRecipe_ExportBusyFlag				: BOOL;
(**)	bManualRecipe_ExportDoneFlag				: BOOL;
(**)	bManualRecipe_ExportErrFlag					: BOOL;
		udManualRecipe_ExportErrId					: UDINT;

